    movel([0.641958, -1.476477, -2.502948, -0.732964, 1.570796, 2.212754],accel_mss,speed_ms,0,blend_radius_m)
    movel([0.641515, -1.476223, -2.503164, -0.733002, 1.570796, 2.212311],accel_mss,speed_ms,0,blend_radius_m)
    movel([0.640075, -1.474344, -2.504756, -0.733289, 1.570796, 2.210872],accel_mss,speed_ms,0,blend_radius_m)
    movel([0.638982, -1.472230, -2.506541, -0.733619, 1.570796, 2.209778],accel_mss,speed_ms,0,blend_radius_m)
    movel([0.638629, -1.472579, -2.506246, -0.733564, 1.570796, 2.209425],accel_mss,speed_ms,0,blend_radius_m)
    movel([0.638365, -1.472967, -2.505919, -0.733503, 1.570796, 2.209162],accel_mss,speed_ms,0,blend_radius_m)
    movel([0.638079, -1.473837, -2.505185, -0.733368, 1.570796, 2.208875],accel_mss,speed_ms,0,blend_radius_m)
    movel([0.638058, -1.474782, -2.504385, -0.733222, 1.570796, 2.208855],accel_mss,speed_ms,0,blend_radius_m)
    movel([0.638230, -1.475759, -2.503558, -0.733073, 1.570796, 2.209026],accel_mss,speed_ms,0,blend_radius_m)
    movel([0.638904, -1.477598, -2.501995, -0.732796, 1.570796, 2.209700],accel_mss,speed_ms,0,blend_radius_m)
    movel([0.639570, -1.478960, -2.500835, -0.732594, 1.570796, 2.210367],accel_mss,speed_ms,0,blend_radius_m)
    movel([0.639752, -1.479499, -2.500375, -0.732515, 1.570796, 2.210548],accel_mss,speed_ms,0,blend_radius_m)
    movel([0.639728, -1.479795, -2.500122, -0.732472, 1.570796, 2.210525],accel_mss,speed_ms,0,blend_radius_m)
    movel([0.639572, -1.480098, -2.499864, -0.732428, 1.570796, 2.210369],accel_mss,speed_ms,0,blend_radius_m)
    movel([0.639281, -1.480378, -2.499624, -0.732387, 1.570796, 2.210078],accel_mss,speed_ms,0,blend_radius_m)
    movel([0.638997, -1.480507, -2.499514, -0.732368, 1.570796, 2.209793],accel_mss,speed_ms,0,blend_radius_m)
    movel([0.638451, -1.480478, -2.499539, -0.732373, 1.570796, 2.209248],accel_mss,speed_ms,0,blend_radius_m)
    movel([0.637722, -1.480353, -2.499646, -0.732391, 1.570796, 2.208518],accel_mss,speed_ms,0,blend_radius_m)
    movel([0.637511, -1.480458, -2.499555, -0.732375, 1.570796, 2.208308],accel_mss,speed_ms,0,blend_radius_m)
    movel([0.637299, -1.480720, -2.499332, -0.732338, 1.570796, 2.208095],accel_mss,speed_ms,0,blend_radius_m)
    movel([0.637184, -1.481038, -2.499059, -0.732292, 1.570796, 2.207981],accel_mss,speed_ms,0,blend_radius_m)
    movel([0.637173, -1.481764, -2.498437, -0.732188, 1.570796, 2.207969],accel_mss,speed_ms,0,blend_radius_m)
    movel([0.637454, -1.483028, -2.497352, -0.732009, 1.570796, 2.208251],accel_mss,speed_ms,0,blend_radius_m)
    movel([0.639119, -1.488150, -2.492930, -0.731309, 1.570796, 2.209915],accel_mss,speed_ms,0,blend_radius_m)
    movel([0.639203, -1.488702, -2.492451, -0.731236, 1.570796, 2.209999],accel_mss,speed_ms,0,blend_radius_m)
    movel([0.639148, -1.489297, -2.491934, -0.731158, 1.570796, 2.209944],accel_mss,speed_ms,0,blend_radius_m)
    movel([0.638894, -1.489854, -2.491449, -0.731086, 1.570796, 2.209690],accel_mss,speed_ms,0,blend_radius_m)
    movel([0.638384, -1.490289, -2.491071, -0.731029, 1.570796, 2.209180],accel_mss,speed_ms,0,blend_radius_m)
    movel([0.637804, -1.490445, -2.490935, -0.731009, 1.570796, 2.208600],accel_mss,speed_ms,0,blend_radius_m)
    movel([0.637303, -1.490327, -2.491037, -0.731024, 1.570796, 2.208099],accel_mss,speed_ms,0,blend_radius_m)
    movel([0.636892, -1.490027, -2.491299, -0.731063, 1.570796, 2.207688],accel_mss,speed_ms,0,blend_radius_m)
    movel([0.636580, -1.489644, -2.491632, -0.731113, 1.570796, 2.207376],accel_mss,speed_ms,0,blend_radius_m)
    movel([0.635083, -1.487144, -2.493802, -0.731443, 1.570796, 2.205879],accel_mss,speed_ms,0,blend_radius_m)
    movel([0.633756, -1.484529, -2.496061, -0.731799, 1.570796, 2.204552],accel_mss,speed_ms,0,blend_radius_m)
    movel([0.632600, -1.481802, -2.498404, -0.732182, 1.570796, 2.203396],accel_mss,speed_ms,0,blend_radius_m)
    movel([0.631623, -1.478968, -2.500828, -0.732593, 1.570796, 2.202419],accel_mss,speed_ms,0,blend_radius_m)
    movel([0.631337, -1.477879, -2.501756, -0.732754, 1.570796, 2.202133],accel_mss,speed_ms,0,blend_radius_m)
    movel([0.631258, -1.476708, -2.502752, -0.732929, 1.570796, 2.202055],accel_mss,speed_ms,0,blend_radius_m)
    movel([0.631373, -1.475970, -2.503379, -0.733040, 1.570796, 2.202169],accel_mss,speed_ms,0,blend_radius_m)
    movel([0.631585, -1.475215, -2.504019, -0.733155, 1.570796, 2.202381],accel_mss,speed_ms,0,blend_radius_m)
    movel([0.632182, -1.473679, -2.505318, -0.733392, 1.570796, 2.202978],accel_mss,speed_ms,0,blend_radius_m)
    movel([0.634868, -1.468171, -2.509946, -0.734271, 1.570796, 2.205664],accel_mss,speed_ms,0,blend_radius_m)
    movel([0.635483, -1.466605, -2.511254, -0.734530, 1.570796, 2.206279],accel_mss,speed_ms,0,blend_radius_m)
    movel([0.635855, -1.465194, -2.512429, -0.734766, 1.570796, 2.206652],accel_mss,speed_ms,0,blend_radius_m)
    movel([0.635914, -1.464584, -2.512936, -0.734870, 1.570796, 2.206711],accel_mss,speed_ms,0,blend_radius_m)
    movel([0.635871, -1.464053, -2.513376, -0.734960, 1.570796, 2.206667],accel_mss,speed_ms,0,blend_radius_m)
    movel([0.635709, -1.463622, -2.513734, -0.735033, 1.570796, 2.206506],accel_mss,speed_ms,0,blend_radius_m)
    movel([0.635418, -1.463300, -2.514000, -0.735088, 1.570796, 2.206215],accel_mss,speed_ms,0,blend_radius_m)
    movel([0.634721, -1.462936, -2.514302, -0.735151, 1.570796, 2.205518],accel_mss,speed_ms,0,blend_radius_m)
    movel([0.634424, -1.462720, -2.514481, -0.735188, 1.570796, 2.205220],accel_mss,speed_ms,0,blend_radius_m)
    movel([0.634271, -1.462407, -2.514740, -0.735242, 1.570796, 2.205068],accel_mss,speed_ms,0,blend_radius_m)
    movel([0.634407, -1.461807, -2.515236, -0.735346, 1.570796, 2.205203],accel_mss,speed_ms,0,blend_radius_m)
    movel([0.634800, -1.461179, -2.515754, -0.735456, 1.570796, 2.205597],accel_mss,speed_ms,0,blend_radius_m)
    movel([0.636148, -1.459190, -2.517393, -0.735807, 1.570796, 2.206945],accel_mss,speed_ms,0,blend_radius_m)
    movel([0.637367, -1.457182, -2.519040, -0.736167, 1.570796, 2.208163],accel_mss,speed_ms,0,blend_radius_m)
    movel([0.639488, -1.453116, -2.522357, -0.736916, 1.570796, 2.210284],accel_mss,speed_ms,0,blend_radius_m)
    movel([0.641323, -1.448978, -2.525707, -0.737704, 1.570796, 2.212119],accel_mss,speed_ms,0,blend_radius_m)
    movel([0.643024, -1.444766, -2.529089, -0.738534, 1.570796, 2.213820],accel_mss,speed_ms,0,blend_radius_m)
    speed_ms = 0.005
    movel([0.643024, -1.436436, -2.525376, -0.750577, 1.570796, 2.213820],accel_mss,speed_ms,0,blend_radius_m)
    speed_ms = 0.040
    movel([0.637764, -1.442161, -2.520832, -0.749396, 1.570796, 2.208560],accel_mss,speed_ms,0,blend_radius_m)
    speed_ms = 0.005
    movel([0.637764, -1.450447, -2.524521, -0.737421, 1.570796, 2.208560],accel_mss,speed_ms,0,blend_radius_m)
    speed_ms = 0.025
    movel([0.634464, -1.454408, -2.521306, -0.736675, 1.570796, 2.205260],accel_mss,speed_ms,0,blend_radius_m)
    movel([0.632715, -1.456330, -2.519737, -0.736322, 1.570796, 2.203511],accel_mss,speed_ms,0,blend_radius_m)
    movel([0.630907, -1.458208, -2.518199, -0.735982, 1.570796, 2.201703],accel_mss,speed_ms,0,blend_radius_m)
    movel([0.630497, -1.456900, -2.519271, -0.736218, 1.570796, 2.201294],accel_mss,speed_ms,0,blend_radius_m)
    movel([0.630400, -1.456693, -2.519440, -0.736256, 1.570796, 2.201197],accel_mss,speed_ms,0,blend_radius_m)
    movel([0.630199, -1.456595, -2.519521, -0.736274, 1.570796, 2.200995],accel_mss,speed_ms,0,blend_radius_m)
    movel([0.629906, -1.456693, -2.519440, -0.736256, 1.570796, 2.200702],accel_mss,speed_ms,0,blend_radius_m)
    movel([0.629627, -1.456902, -2.519269, -0.736218, 1.570796, 2.200423],accel_mss,speed_ms,0,blend_radius_m)
    movel([0.627898, -1.458194, -2.518210, -0.735985, 1.570796, 2.198694],accel_mss,speed_ms,0,blend_radius_m)
    movel([0.626047, -1.459278, -2.517320, -0.735791, 1.570796, 2.196843],accel_mss,speed_ms,0,blend_radius_m)
    movel([0.625596, -1.459460, -2.517171, -0.735759, 1.570796, 2.196392],accel_mss,speed_ms,0,blend_radius_m)
    movel([0.625231, -1.459431, -2.517194, -0.735764, 1.570796, 2.196027],accel_mss,speed_ms,0,blend_radius_m)
    movel([0.625146, -1.459173, -2.517406, -0.735810, 1.570796, 2.195943],accel_mss,speed_ms,0,blend_radius_m)
    movel([0.625241, -1.458837, -2.517683, -0.735870, 1.570796, 2.196037],accel_mss,speed_ms,0,blend_radius_m)
    movel([0.626199, -1.456787, -2.519363, -0.736239, 1.570796, 2.196995],accel_mss,speed_ms,0,blend_radius_m)
    movel([0.627476, -1.454770, -2.521011, -0.736608, 1.570796, 2.198272],accel_mss,speed_ms,0,blend_radius_m)
    speed_ms = 0.005
    movel([0.627476, -1.446519, -2.517340, -0.748530, 1.570796, 2.198272],accel_mss,speed_ms,0,blend_radius_m)
    speed_ms = 0.040
    movel([0.627988, -1.451771, -2.513092, -0.747526, 1.570796, 2.198784],accel_mss,speed_ms,0,blend_radius_m)
    speed_ms = 0.005
    movel([0.627988, -1.459981, -2.516742, -0.735666, 1.570796, 2.198784],accel_mss,speed_ms,0,blend_radius_m)
    speed_ms = 0.025
    movel([0.626151, -1.462942, -2.514297, -0.735150, 1.570796, 2.196948],accel_mss,speed_ms,0,blend_radius_m)
    movel([0.625097, -1.464385, -2.513101, -0.734903, 1.570796, 2.195893],accel_mss,speed_ms,0,blend_radius_m)
    movel([0.622748, -1.467165, -2.510787, -0.734437, 1.570796, 2.193545],accel_mss,speed_ms,0,blend_radius_m)
    movel([0.621462, -1.468491, -2.509679, -0.734219, 1.570796, 2.192259],accel_mss,speed_ms,0,blend_radius_m)
    movel([0.618694, -1.470988, -2.507585, -0.733816, 1.570796, 2.189491],accel_mss,speed_ms,0,blend_radius_m)
    movel([0.619378, -1.470024, -2.508394, -0.733970, 1.570796, 2.190174],accel_mss,speed_ms,0,blend_radius_m)
    movel([0.619797, -1.469022, -2.509234, -0.734132, 1.570796, 2.190594],accel_mss,speed_ms,0,blend_radius_m)
    movel([0.619930, -1.468054, -2.510045, -0.734291, 1.570796, 2.190726],accel_mss,speed_ms,0,blend_radius_m)
    movel([0.619753, -1.467190, -2.510766, -0.734433, 1.570796, 2.190549],accel_mss,speed_ms,0,blend_radius_m)
    speed_ms = 0.005
    movel([0.619753, -1.459037, -2.507146, -0.746205, 1.570796, 2.190549],accel_mss,speed_ms,0,blend_radius_m)
    speed_ms = 0.040
    movel([0.608750, -1.458273, -2.507776, -0.746340, 1.570796, 2.179546],accel_mss,speed_ms,0,blend_radius_m)
    speed_ms = 0.005
    movel([0.608750, -1.466431, -2.511399, -0.734559, 1.570796, 2.179546],accel_mss,speed_ms,0,blend_radius_m)
    speed_ms = 0.025
    movel([0.606276, -1.467605, -2.510420, -0.734364, 1.570796, 2.177072],accel_mss,speed_ms,0,blend_radius_m)
    movel([0.603766, -1.468519, -2.509656, -0.734215, 1.570796, 2.174563],accel_mss,speed_ms,0,blend_radius_m)
    movel([0.601263, -1.469162, -2.509117, -0.734110, 1.570796, 2.172059],accel_mss,speed_ms,0,blend_radius_m)
    movel([0.598809, -1.469521, -2.508816, -0.734051, 1.570796, 2.169605],accel_mss,speed_ms,0,blend_radius_m)
    movel([0.599716, -1.468751, -2.509462, -0.734177, 1.570796, 2.170512],accel_mss,speed_ms,0,blend_radius_m)
    movel([0.600486, -1.467955, -2.510127, -0.734307, 1.570796, 2.171283],accel_mss,speed_ms,0,blend_radius_m)
    movel([0.601057, -1.467211, -2.510748, -0.734429, 1.570796, 2.171853],accel_mss,speed_ms,0,blend_radius_m)
    movel([0.601366, -1.466593, -2.511264, -0.734532, 1.570796, 2.172162],accel_mss,speed_ms,0,blend_radius_m)
    movel([0.601345, -1.466181, -2.511607, -0.734601, 1.570796, 2.172142],accel_mss,speed_ms,0,blend_radius_m)
    movel([0.601194, -1.466075, -2.511695, -0.734618, 1.570796, 2.171990],accel_mss,speed_ms,0,blend_radius_m)
    movel([0.600934, -1.466048, -2.511718, -0.734623, 1.570796, 2.171730],accel_mss,speed_ms,0,blend_radius_m)
    movel([0.600067, -1.466274, -2.511529, -0.734585, 1.570796, 2.170864],accel_mss,speed_ms,0,blend_radius_m)
    movel([0.597596, -1.467480, -2.510524, -0.734385, 1.570796, 2.168392],accel_mss,speed_ms,0,blend_radius_m)
    movel([0.596477, -1.467956, -2.510126, -0.734307, 1.570796, 2.167273],accel_mss,speed_ms,0,blend_radius_m)
    movel([0.594203, -1.468674, -2.509526, -0.734189, 1.570796, 2.164999],accel_mss,speed_ms,0,blend_radius_m)
    movel([0.593077, -1.468905, -2.509333, -0.734152, 1.570796, 2.163873],accel_mss,speed_ms,0,blend_radius_m)
    movel([0.591978, -1.469037, -2.509222, -0.734130, 1.570796, 2.162775],accel_mss,speed_ms,0,blend_radius_m)
    movel([0.590919, -1.469071, -2.509194, -0.734125, 1.570796, 2.161716],accel_mss,speed_ms,0,blend_radius_m)
    movel([0.589919, -1.468994, -2.509258, -0.734137, 1.570796, 2.160715],accel_mss,speed_ms,0,blend_radius_m)
    movel([0.591630, -1.468026, -2.510068, -0.734295, 1.570796, 2.162426],accel_mss,speed_ms,0,blend_radius_m)
    movel([0.593324, -1.467014, -2.510913, -0.734462, 1.570796, 2.164121],accel_mss,speed_ms,0,blend_radius_m)
    movel([0.594264, -1.466177, -2.511611, -0.734601, 1.570796, 2.165060],accel_mss,speed_ms,0,blend_radius_m)
    movel([0.595003, -1.465226, -2.512402, -0.734761, 1.570796, 2.165799],accel_mss,speed_ms,0,blend_radius_m)
    movel([0.595149, -1.464828, -2.512733, -0.734828, 1.570796, 2.165945],accel_mss,speed_ms,0,blend_radius_m)
    movel([0.595062, -1.464545, -2.512968, -0.734876, 1.570796, 2.165858],accel_mss,speed_ms,0,blend_radius_m)
    movel([0.594686, -1.464428, -2.513065, -0.734896, 1.570796, 2.165483],accel_mss,speed_ms,0,blend_radius_m)
    movel([0.593960, -1.464526, -2.512983, -0.734879, 1.570796, 2.164756],accel_mss,speed_ms,0,blend_radius_m)
    movel([0.589880, -1.465593, -2.512097, -0.734699, 1.570796, 2.160677],accel_mss,speed_ms,0,blend_radius_m)
    movel([0.587928, -1.465897, -2.511843, -0.734648, 1.570796, 2.158724],accel_mss,speed_ms,0,blend_radius_m)
    movel([0.587015, -1.465903, -2.511839, -0.734647, 1.570796, 2.157811],accel_mss,speed_ms,0,blend_radius_m)
    movel([0.586157, -1.465776, -2.511945, -0.734669, 1.570796, 2.156953],accel_mss,speed_ms,0,blend_radius_m)
    speed_ms = 0.005
    movel([0.586157, -1.457612, -2.508319, -0.746458, 1.570796, 2.156953],accel_mss,speed_ms,0,blend_radius_m)
    speed_ms = 0.040
    movel([0.608445, -1.444545, -2.518925, -0.748919, 1.570796, 2.179242],accel_mss,speed_ms,0,blend_radius_m)
    speed_ms = 0.005
    movel([0.608445, -1.452812, -2.522604, -0.736973, 1.570796, 2.179242],accel_mss,speed_ms,0,blend_radius_m)
    speed_ms = 0.025
    movel([0.609102, -1.451455, -2.523704, -0.737229, 1.570796, 2.179898],accel_mss,speed_ms,0,blend_radius_m)
    movel([0.610004, -1.450153, -2.524759, -0.737478, 1.570796, 2.180800],accel_mss,speed_ms,0,blend_radius_m)
    movel([0.611115, -1.448916, -2.525757, -0.737716, 1.570796, 2.181912],accel_mss,speed_ms,0,blend_radius_m)
    movel([0.612394, -1.447766, -2.526683, -0.737940, 1.570796, 2.183190],accel_mss,speed_ms,0,blend_radius_m)
    movel([0.613809, -1.446716, -2.527526, -0.738146, 1.570796, 2.184605],accel_mss,speed_ms,0,blend_radius_m)
    movel([0.615315, -1.445789, -2.528270, -0.738330, 1.570796, 2.186111],accel_mss,speed_ms,0,blend_radius_m)
    movel([0.616882, -1.444997, -2.528905, -0.738488, 1.570796, 2.187678],accel_mss,speed_ms,0,blend_radius_m)
    movel([0.618464, -1.444359, -2.529414, -0.738615, 1.570796, 2.189261],accel_mss,speed_ms,0,blend_radius_m)
    movel([0.620408, -1.443761, -2.529892, -0.738736, 1.570796, 2.191205],accel_mss,speed_ms,0,blend_radius_m)
    movel([0.624291, -1.442705, -2.530734, -0.738950, 1.570796, 2.195087],accel_mss,speed_ms,0,blend_radius_m)
    movel([0.626231, -1.442020, -2.531280, -0.739089, 1.570796, 2.197028],accel_mss,speed_ms,0,blend_radius_m)
    movel([0.628170, -1.441040, -2.532058, -0.739290, 1.570796, 2.198966],accel_mss,speed_ms,0,blend_radius_m)
    movel([0.629096, -1.440430, -2.532542, -0.739416, 1.570796, 2.199893],accel_mss,speed_ms,0,blend_radius_m)
    movel([0.629958, -1.439753, -2.533079, -0.739557, 1.570796, 2.200754],accel_mss,speed_ms,0,blend_radius_m)
    movel([0.630728, -1.439017, -2.533662, -0.739710, 1.570796, 2.201524],accel_mss,speed_ms,0,blend_radius_m)
    movel([0.631381, -1.438234, -2.534281, -0.739874, 1.570796, 2.202177],accel_mss,speed_ms,0,blend_radius_m)
    movel([0.631884, -1.437414, -2.534928, -0.740047, 1.570796, 2.202680],accel_mss,speed_ms,0,blend_radius_m)
    movel([0.632210, -1.436568, -2.535594, -0.740227, 1.570796, 2.203006],accel_mss,speed_ms,0,blend_radius_m)
    speed_ms = 0.005
    movel([0.632210, -1.428174, -2.531847, -0.752368, 1.570796, 2.203006],accel_mss,speed_ms,0,blend_radius_m)
    speed_ms = 0.040
    movel([0.634472, -1.421241, -2.537198, -0.753950, 1.570796, 2.205268],accel_mss,speed_ms,0,blend_radius_m)
    speed_ms = 0.005
    movel([0.634472, -1.429688, -2.540974, -0.741726, 1.570796, 2.205268],accel_mss,speed_ms,0,blend_radius_m)
    speed_ms = 0.025
    movel([0.630966, -1.434319, -2.537361, -0.740709, 1.570796, 2.201762],accel_mss,speed_ms,0,blend_radius_m)
    movel([0.630012, -1.435247, -2.536633, -0.740509, 1.570796, 2.200808],accel_mss,speed_ms,0,blend_radius_m)
    movel([0.628877, -1.435944, -2.536085, -0.740360, 1.570796, 2.199673],accel_mss,speed_ms,0,blend_radius_m)
    movel([0.627663, -1.436404, -2.535723, -0.740262, 1.570796, 2.198460],accel_mss,speed_ms,0,blend_radius_m)
    movel([0.623784, -1.437426, -2.534919, -0.740045, 1.570796, 2.194581],accel_mss,speed_ms,0,blend_radius_m)
    movel([0.622396, -1.437944, -2.534510, -0.739935, 1.570796, 2.193193],accel_mss,speed_ms,0,blend_radius_m)
    movel([0.621022, -1.438571, -2.534015, -0.739804, 1.570796, 2.191818],accel_mss,speed_ms,0,blend_radius_m)
    movel([0.619676, -1.439294, -2.533443, -0.739652, 1.570796, 2.190472],accel_mss,speed_ms,0,blend_radius_m)
    movel([0.618436, -1.440141, -2.532772, -0.739476, 1.570796, 2.189232],accel_mss,speed_ms,0,blend_radius_m)
    movel([0.617280, -1.441094, -2.532016, -0.739279, 1.570796, 2.188076],accel_mss,speed_ms,0,blend_radius_m)
    movel([0.616136, -1.442049, -2.531256, -0.739083, 1.570796, 2.186932],accel_mss,speed_ms,0,blend_radius_m)
    movel([0.614930, -1.442905, -2.530575, -0.738909, 1.570796, 2.185726],accel_mss,speed_ms,0,blend_radius_m)
    movel([0.615593, -1.439744, -2.533086, -0.739559, 1.570796, 2.186390],accel_mss,speed_ms,0,blend_radius_m)
    movel([0.616059, -1.438916, -2.533742, -0.739731, 1.570796, 2.186855],accel_mss,speed_ms,0,blend_radius_m)
    movel([0.616636, -1.438140, -2.534355, -0.739894, 1.570796, 2.187432],accel_mss,speed_ms,0,blend_radius_m)
    movel([0.617323, -1.437413, -2.534928, -0.740047, 1.570796, 2.188119],accel_mss,speed_ms,0,blend_radius_m)
    movel([0.618129, -1.436734, -2.535464, -0.740191, 1.570796, 2.188926],accel_mss,speed_ms,0,blend_radius_m)
    movel([0.619413, -1.435981, -2.536056, -0.740352, 1.570796, 2.190209],accel_mss,speed_ms,0,blend_radius_m)
    movel([0.621123, -1.435253, -2.536628, -0.740508, 1.570796, 2.191920],accel_mss,speed_ms,0,blend_radius_m)
    movel([0.625153, -1.433842, -2.537735, -0.740812, 1.570796, 2.195949],accel_mss,speed_ms,0,blend_radius_m)
    movel([0.627133, -1.433147, -2.538278, -0.740963, 1.570796, 2.197930],accel_mss,speed_ms,0,blend_radius_m)
    movel([0.628867, -1.432445, -2.538827, -0.741117, 1.570796, 2.199663],accel_mss,speed_ms,0,blend_radius_m)
    movel([0.630181, -1.431732, -2.539383, -0.741273, 1.570796, 2.200977],accel_mss,speed_ms,0,blend_radius_m)
    movel([0.630630, -1.431367, -2.539668, -0.741354, 1.570796, 2.201426],accel_mss,speed_ms,0,blend_radius_m)
    movel([0.630911, -1.430993, -2.539959, -0.741436, 1.570796, 2.201707],accel_mss,speed_ms,0,blend_radius_m)
    speed_ms = 0.005
    movel([0.630911, -1.422556, -2.536188, -0.753645, 1.570796, 2.201707],accel_mss,speed_ms,0,blend_radius_m)
    speed_ms = 0.040
    movel([0.626406, -1.418603, -2.539215, -0.754571, 1.570796, 2.197203],accel_mss,speed_ms,0,blend_radius_m)
    speed_ms = 0.005
    movel([0.626406, -1.427071, -2.543002, -0.742316, 1.570796, 2.197203],accel_mss,speed_ms,0,blend_radius_m)
    speed_ms = 0.025
    movel([0.625978, -1.426676, -2.543308, -0.742406, 1.570796, 2.196775],accel_mss,speed_ms,0,blend_radius_m)
    movel([0.625701, -1.426178, -2.543692, -0.742519, 1.570796, 2.196497],accel_mss,speed_ms,0,blend_radius_m)
    movel([0.625515, -1.424957, -2.544632, -0.742799, 1.570796, 2.196311],accel_mss,speed_ms,0,blend_radius_m)
    movel([0.625692, -1.423549, -2.545715, -0.743125, 1.570796, 2.196488],accel_mss,speed_ms,0,blend_radius_m)
    movel([0.626077, -1.422092, -2.546832, -0.743466, 1.570796, 2.196873],accel_mss,speed_ms,0,blend_radius_m)
    movel([0.626302, -1.421561, -2.547237, -0.743590, 1.570796, 2.197098],accel_mss,speed_ms,0,blend_radius_m)
    movel([0.627024, -1.420869, -2.547766, -0.743754, 1.570796, 2.197820],accel_mss,speed_ms,0,blend_radius_m)
    movel([0.629266, -1.419088, -2.549123, -0.744177, 1.570796, 2.200063],accel_mss,speed_ms,0,blend_radius_m)
    movel([0.633612, -1.415346, -2.551960, -0.745083, 1.570796, 2.204409],accel_mss,speed_ms,0,blend_radius_m)
    movel([0.635707, -1.413393, -2.553432, -0.745564, 1.570796, 2.206503],accel_mss,speed_ms,0,blend_radius_m)
    speed_ms = 0.005
    movel([0.635707, -1.404821, -2.549586, -0.757982, 1.570796, 2.206503],accel_mss,speed_ms,0,blend_radius_m)
    speed_ms = 0.040
    movel([0.631730, -1.404605, -2.549746, -0.758038, 1.570796, 2.202526],accel_mss,speed_ms,0,blend_radius_m)
    speed_ms = 0.005
    movel([0.631730, -1.413178, -2.553593, -0.745617, 1.570796, 2.202526],accel_mss,speed_ms,0,blend_radius_m)
    speed_ms = 0.025
    movel([0.630561, -1.414434, -2.552648, -0.745307, 1.570796, 2.201357],accel_mss,speed_ms,0,blend_radius_m)
    movel([0.629275, -1.415602, -2.551767, -0.745021, 1.570796, 2.200071],accel_mss,speed_ms,0,blend_radius_m)
    movel([0.627884, -1.416569, -2.551035, -0.744785, 1.570796, 2.198680],accel_mss,speed_ms,0,blend_radius_m)
    movel([0.627150, -1.416945, -2.550750, -0.744694, 1.570796, 2.197947],accel_mss,speed_ms,0,blend_radius_m)
    movel([0.625657, -1.417523, -2.550312, -0.744554, 1.570796, 2.196453],accel_mss,speed_ms,0,blend_radius_m)
    movel([0.625143, -1.417996, -2.549953, -0.744440, 1.570796, 2.195940],accel_mss,speed_ms,0,blend_radius_m)
    movel([0.621578, -1.421930, -2.546956, -0.743504, 1.570796, 2.192374],accel_mss,speed_ms,0,blend_radius_m)
    movel([0.621243, -1.422316, -2.546660, -0.743413, 1.570796, 2.192039],accel_mss,speed_ms,0,blend_radius_m)
    movel([0.621016, -1.422721, -2.546349, -0.743318, 1.570796, 2.191812],accel_mss,speed_ms,0,blend_radius_m)
    movel([0.621038, -1.423264, -2.545933, -0.743192, 1.570796, 2.191834],accel_mss,speed_ms,0,blend_radius_m)
    movel([0.621320, -1.423696, -2.545602, -0.743091, 1.570796, 2.192117],accel_mss,speed_ms,0,blend_radius_m)
    movel([0.622190, -1.424884, -2.544689, -0.742816, 1.570796, 2.192987],accel_mss,speed_ms,0,blend_radius_m)
    movel([0.622880, -1.426189, -2.543683, -0.742517, 1.570796, 2.193677],accel_mss,speed_ms,0,blend_radius_m)
    movel([0.623286, -1.427633, -2.542568, -0.742188, 1.570796, 2.194082],accel_mss,speed_ms,0,blend_radius_m)
    movel([0.623292, -1.429238, -2.541324, -0.741827, 1.570796, 2.194088],accel_mss,speed_ms,0,blend_radius_m)
    speed_ms = 0.005
    movel([0.623292, -1.420787, -2.537546, -0.754056, 1.570796, 2.194088],accel_mss,speed_ms,0,blend_radius_m)
    speed_ms = 0.040
    movel([0.614239, -1.430940, -2.529692, -0.751757, 1.570796, 2.185036],accel_mss,speed_ms,0,blend_radius_m)
    speed_ms = 0.005
    movel([0.614239, -1.439312, -2.533428, -0.739649, 1.570796, 2.185036],accel_mss,speed_ms,0,blend_radius_m)
    speed_ms = 0.025
    movel([0.613899, -1.439397, -2.533361, -0.739631, 1.570796, 2.184695],accel_mss,speed_ms,0,blend_radius_m)
    movel([0.613539, -1.439584, -2.533213, -0.739592, 1.570796, 2.184336],accel_mss,speed_ms,0,blend_radius_m)
    movel([0.611897, -1.440794, -2.532254, -0.739341, 1.570796, 2.182693],accel_mss,speed_ms,0,blend_radius_m)
    movel([0.611689, -1.440847, -2.532211, -0.739330, 1.570796, 2.182486],accel_mss,speed_ms,0,blend_radius_m)
    movel([0.611472, -1.440734, -2.532301, -0.739353, 1.570796, 2.182269],accel_mss,speed_ms,0,blend_radius_m)
    movel([0.611391, -1.440464, -2.532516, -0.739409, 1.570796, 2.182188],accel_mss,speed_ms,0,blend_radius_m)
    movel([0.611527, -1.439641, -2.533168, -0.739580, 1.570796, 2.182323],accel_mss,speed_ms,0,blend_radius_m)
    movel([0.612164, -1.438124, -2.534368, -0.739897, 1.570796, 2.182960],accel_mss,speed_ms,0,blend_radius_m)
    movel([0.613130, -1.436783, -2.535425, -0.740181, 1.570796, 2.183926],accel_mss,speed_ms,0,blend_radius_m)
    movel([0.614280, -1.435499, -2.536435, -0.740455, 1.570796, 2.185077],accel_mss,speed_ms,0,blend_radius_m)
    movel([0.615503, -1.434287, -2.537386, -0.740716, 1.570796, 2.186300],accel_mss,speed_ms,0,blend_radius_m)
    movel([0.616788, -1.433202, -2.538236, -0.740951, 1.570796, 2.187584],accel_mss,speed_ms,0,blend_radius_m)
    movel([0.618128, -1.432240, -2.538987, -0.741162, 1.570796, 2.188924],accel_mss,speed_ms,0,blend_radius_m)
    movel([0.619521, -1.431398, -2.539644, -0.741347, 1.570796, 2.190317],accel_mss,speed_ms,0,blend_radius_m)
    movel([0.620965, -1.430671, -2.540210, -0.741508, 1.570796, 2.191761],accel_mss,speed_ms,0,blend_radius_m)
    movel([0.622453, -1.430055, -2.540689, -0.741644, 1.570796, 2.193249],accel_mss,speed_ms,0,blend_radius_m)
    movel([0.623986, -1.429546, -2.541085, -0.741758, 1.570796, 2.194782],accel_mss,speed_ms,0,blend_radius_m)
    movel([0.625558, -1.429138, -2.541401, -0.741849, 1.570796, 2.196355],accel_mss,speed_ms,0,blend_radius_m)
    movel([0.627800, -1.428405, -2.541970, -0.742014, 1.570796, 2.198597],accel_mss,speed_ms,0,blend_radius_m)
    movel([0.630263, -1.427347, -2.542789, -0.742253, 1.570796, 2.201059],accel_mss,speed_ms,0,blend_radius_m)
    movel([0.632999, -1.425997, -2.543831, -0.742561, 1.570796, 2.203795],accel_mss,speed_ms,0,blend_radius_m)
    speed_ms = 0.005
    movel([0.632999, -1.417521, -2.540039, -0.754829, 1.570796, 2.203795],accel_mss,speed_ms,0,blend_radius_m)
    speed_ms = 0.040
    movel([0.631529, -1.416683, -2.540677, -0.755030, 1.570796, 2.202326],accel_mss,speed_ms,0,blend_radius_m)
    speed_ms = 0.005
    movel([0.631529, -1.425165, -2.544473, -0.742752, 1.570796, 2.202326],accel_mss,speed_ms,0,blend_radius_m)
    speed_ms = 0.025
    movel([0.634472, -1.422332, -2.546648, -0.743409, 1.570796, 2.205269],accel_mss,speed_ms,0,blend_radius_m)
    movel([0.637560, -1.419600, -2.548734, -0.744055, 1.570796, 2.208356],accel_mss,speed_ms,0,blend_radius_m)
    movel([0.639176, -1.418327, -2.549702, -0.744360, 1.570796, 2.209972],accel_mss,speed_ms,0,blend_radius_m)
    movel([0.640843, -1.417142, -2.550601, -0.744646, 1.570796, 2.211640],accel_mss,speed_ms,0,blend_radius_m)
    movel([0.642574, -1.416069, -2.551413, -0.744907, 1.570796, 2.213371],accel_mss,speed_ms,0,blend_radius_m)
    movel([0.644367, -1.415131, -2.552122, -0.745136, 1.570796, 2.215163],accel_mss,speed_ms,0,blend_radius_m)
    movel([0.649060, -1.413130, -2.553629, -0.745629, 1.570796, 2.219856],accel_mss,speed_ms,0,blend_radius_m)
    movel([0.651133, -1.412130, -2.554381, -0.745878, 1.570796, 2.221930],accel_mss,speed_ms,0,blend_radius_m)
    movel([0.652150, -1.411557, -2.554810, -0.746021, 1.570796, 2.222947],accel_mss,speed_ms,0,blend_radius_m)
    movel([0.653131, -1.410897, -2.555305, -0.746187, 1.570796, 2.223928],accel_mss,speed_ms,0,blend_radius_m)
    movel([0.655731, -1.408453, -2.557129, -0.746806, 1.570796, 2.226527],accel_mss,speed_ms,0,blend_radius_m)
    speed_ms = 0.005
    movel([0.655731, -1.399844, -2.553262, -0.759283, 1.570796, 2.226527],accel_mss,speed_ms,0,blend_radius_m)
    speed_ms = 0.040
    movel([0.661836, -1.394252, -2.557350, -0.760788, 1.570796, 2.232632],accel_mss,speed_ms,0,blend_radius_m)
    speed_ms = 0.005
    movel([0.661836, -1.402902, -2.561241, -0.748245, 1.570796, 2.232632],accel_mss,speed_ms,0,blend_radius_m)
    speed_ms = 0.025
    movel([0.663890, -1.400838, -2.562759, -0.748792, 1.570796, 2.234687],accel_mss,speed_ms,0,blend_radius_m)
    movel([0.665035, -1.399965, -2.563398, -0.749025, 1.570796, 2.235831],accel_mss,speed_ms,0,blend_radius_m)
    movel([0.666278, -1.399312, -2.563877, -0.749200, 1.570796, 2.237075],accel_mss,speed_ms,0,blend_radius_m)
    movel([0.667177, -1.399037, -2.564078, -0.749274, 1.570796, 2.237974],accel_mss,speed_ms,0,blend_radius_m)
    movel([0.668058, -1.398894, -2.564182, -0.749313, 1.570796, 2.238854],accel_mss,speed_ms,0,blend_radius_m)
    movel([0.669780, -1.398801, -2.564250, -0.749338, 1.570796, 2.240576],accel_mss,speed_ms,0,blend_radius_m)
    movel([0.671376, -1.398578, -2.564413, -0.749398, 1.570796, 2.242173],accel_mss,speed_ms,0,blend_radius_m)
    movel([0.672788, -1.398079, -2.564777, -0.749533, 1.570796, 2.243584],accel_mss,speed_ms,0,blend_radius_m)
    movel([0.675757, -1.396456, -2.565959, -0.749974, 1.570796, 2.246553],accel_mss,speed_ms,0,blend_radius_m)
    movel([0.676370, -1.396174, -2.566165, -0.750051, 1.570796, 2.247166],accel_mss,speed_ms,0,blend_radius_m)
    movel([0.676978, -1.396006, -2.566287, -0.750097, 1.570796, 2.247775],accel_mss,speed_ms,0,blend_radius_m)
    movel([0.678181, -1.395918, -2.566350, -0.750121, 1.570796, 2.248978],accel_mss,speed_ms,0,blend_radius_m)
    movel([0.680510, -1.396020, -2.566276, -0.750093, 1.570796, 2.251307],accel_mss,speed_ms,0,blend_radius_m)
    movel([0.683082, -1.395846, -2.566403, -0.750140, 1.570796, 2.253879],accel_mss,speed_ms,0,blend_radius_m)
    movel([0.684409, -1.395623, -2.566565, -0.750202, 1.570796, 2.255205],accel_mss,speed_ms,0,blend_radius_m)
    movel([0.685767, -1.395218, -2.566859, -0.750313, 1.570796, 2.256564],accel_mss,speed_ms,0,blend_radius_m)
    movel([0.686865, -1.394669, -2.567256, -0.750464, 1.570796, 2.257661],accel_mss,speed_ms,0,blend_radius_m)
    movel([0.687861, -1.393908, -2.567807, -0.750674, 1.570796, 2.258657],accel_mss,speed_ms,0,blend_radius_m)
    movel([0.688550, -1.393039, -2.568435, -0.750915, 1.570796, 2.259346],accel_mss,speed_ms,0,blend_radius_m)
    movel([0.688714, -1.392599, -2.568753, -0.751037, 1.570796, 2.259510],accel_mss,speed_ms,0,blend_radius_m)
    movel([0.688723, -1.392174, -2.569060, -0.751156, 1.570796, 2.259519],accel_mss,speed_ms,0,blend_radius_m)
    movel([0.688416, -1.391422, -2.569601, -0.751366, 1.570796, 2.259212],accel_mss,speed_ms,0,blend_radius_m)
    movel([0.687831, -1.390766, -2.570073, -0.751550, 1.570796, 2.258627],accel_mss,speed_ms,0,blend_radius_m)
    movel([0.687019, -1.390220, -2.570465, -0.751704, 1.570796, 2.257815],accel_mss,speed_ms,0,blend_radius_m)
    movel([0.686046, -1.389794, -2.570771, -0.751824, 1.570796, 2.256842],accel_mss,speed_ms,0,blend_radius_m)
    movel([0.684965, -1.389510, -2.570975, -0.751904, 1.570796, 2.255761],accel_mss,speed_ms,0,blend_radius_m)
    movel([0.683839, -1.389375, -2.571072, -0.751943, 1.570796, 2.254635],accel_mss,speed_ms,0,blend_radius_m)
    movel([0.682724, -1.389408, -2.571048, -0.751933, 1.570796, 2.253520],accel_mss,speed_ms,0,blend_radius_m)
    movel([0.681679, -1.389620, -2.570896, -0.751873, 1.570796, 2.252475],accel_mss,speed_ms,0,blend_radius_m)
    movel([0.680107, -1.390284, -2.570419, -0.751686, 1.570796, 2.250903],accel_mss,speed_ms,0,blend_radius_m)
    movel([0.675473, -1.392714, -2.568670, -0.751005, 1.570796, 2.246269],accel_mss,speed_ms,0,blend_radius_m)
    movel([0.672351, -1.394092, -2.567674, -0.750623, 1.570796, 2.243147],accel_mss,speed_ms,0,blend_radius_m)
    movel([0.669641, -1.394935, -2.567064, -0.750390, 1.570796, 2.240437],accel_mss,speed_ms,0,blend_radius_m)
    movel([0.668305, -1.395322, -2.566783, -0.750284, 1.570796, 2.239101],accel_mss,speed_ms,0,blend_radius_m)
    movel([0.666980, -1.395830, -2.566414, -0.750145, 1.570796, 2.237776],accel_mss,speed_ms,0,blend_radius_m)
    movel([0.665633, -1.396532, -2.565904, -0.749953, 1.570796, 2.236430],accel_mss,speed_ms,0,blend_radius_m)
    movel([0.664346, -1.397350, -2.565309, -0.749730, 1.570796, 2.235142],accel_mss,speed_ms,0,blend_radius_m)
    movel([0.663112, -1.398265, -2.564641, -0.749482, 1.570796, 2.233909],accel_mss,speed_ms,0,blend_radius_m)
    movel([0.661932, -1.399254, -2.563919, -0.749216, 1.570796, 2.232728],accel_mss,speed_ms,0,blend_radius_m)
    movel([0.659712, -1.401374, -2.562365, -0.748649, 1.570796, 2.230508],accel_mss,speed_ms,0,blend_radius_m)
    movel([0.657647, -1.403546, -2.560767, -0.748076, 1.570796, 2.228444],accel_mss,speed_ms,0,blend_radius_m)
    speed_ms = 0.005
    movel([0.657647, -1.394900, -2.556878, -0.760611, 1.570796, 2.228444],accel_mss,speed_ms,0,blend_radius_m)
    speed_ms = 0.040
    movel([0.654415, -1.395213, -2.556651, -0.760526, 1.570796, 2.225212],accel_mss,speed_ms,0,blend_radius_m)
    speed_ms = 0.005
    movel([0.654415, -1.403856, -2.560538, -0.747995, 1.570796, 2.225212],accel_mss,speed_ms,0,blend_radius_m)
    speed_ms = 0.025
    movel([0.657764, -1.400491, -2.563013, -0.748885, 1.570796, 2.228560],accel_mss,speed_ms,0,blend_radius_m)
    movel([0.659213, -1.399123, -2.564014, -0.749251, 1.570796, 2.230010],accel_mss,speed_ms,0,blend_radius_m)
    movel([0.660598, -1.397708, -2.565048, -0.749633, 1.570796, 2.231394],accel_mss,speed_ms,0,blend_radius_m)
    movel([0.661658, -1.396409, -2.565994, -0.749987, 1.570796, 2.232454],accel_mss,speed_ms,0,blend_radius_m)
    movel([0.662556, -1.395052, -2.566979, -0.750358, 1.570796, 2.233353],accel_mss,speed_ms,0,blend_radius_m)
    movel([0.663277, -1.393664, -2.567984, -0.750741, 1.570796, 2.234073],accel_mss,speed_ms,0,blend_radius_m)
    movel([0.663803, -1.392274, -2.568987, -0.751128, 1.570796, 2.234600],accel_mss,speed_ms,0,blend_radius_m)
    movel([0.664421, -1.392300, -2.568969, -0.751120, 1.570796, 2.235217],accel_mss,speed_ms,0,blend_radius_m)
    movel([0.664952, -1.392477, -2.568841, -0.751071, 1.570796, 2.235749],accel_mss,speed_ms,0,blend_radius_m)
    movel([0.665902, -1.393010, -2.568456, -0.750923, 1.570796, 2.236698],accel_mss,speed_ms,0,blend_radius_m)
    movel([0.666957, -1.393447, -2.568141, -0.750801, 1.570796, 2.237753],accel_mss,speed_ms,0,blend_radius_m)
    movel([0.667567, -1.393492, -2.568108, -0.750789, 1.570796, 2.238364],accel_mss,speed_ms,0,blend_radius_m)
    movel([0.668235, -1.393324, -2.568229, -0.750835, 1.570796, 2.239032],accel_mss,speed_ms,0,blend_radius_m)
    movel([0.676287, -1.390042, -2.570593, -0.751754, 1.570796, 2.247083],accel_mss,speed_ms,0,blend_radius_m)
    movel([0.676745, -1.389077, -2.571285, -0.752027, 1.570796, 2.247541],accel_mss,speed_ms,0,blend_radius_m)
    movel([0.676931, -1.388102, -2.571983, -0.752304, 1.570796, 2.247728],accel_mss,speed_ms,0,blend_radius_m)
    movel([0.676838, -1.387168, -2.572650, -0.752571, 1.570796, 2.247634],accel_mss,speed_ms,0,blend_radius_m)
    movel([0.676462, -1.386329, -2.573248, -0.752812, 1.570796, 2.247259],accel_mss,speed_ms,0,blend_radius_m)
    movel([0.677727, -1.386688, -2.572992, -0.752709, 1.570796, 2.248523],accel_mss,speed_ms,0,blend_radius_m)
    movel([0.678785, -1.387289, -2.572563, -0.752536, 1.570796, 2.249582],accel_mss,speed_ms,0,blend_radius_m)
    movel([0.679587, -1.388095, -2.571987, -0.752306, 1.570796, 2.250383],accel_mss,speed_ms,0,blend_radius_m)
    movel([0.680086, -1.389070, -2.571290, -0.752029, 1.570796, 2.250882],accel_mss,speed_ms,0,blend_radius_m)
    speed_ms = 0.005
    movel([0.680086, -1.380317, -2.567338, -0.764734, 1.570796, 2.250882],accel_mss,speed_ms,0,blend_radius_m)
    speed_ms = 0.040
    movel([0.682625, -1.376904, -2.569742, -0.765743, 1.570796, 2.253421],accel_mss,speed_ms,0,blend_radius_m)
    speed_ms = 0.005
    movel([0.682625, -1.385682, -2.573709, -0.752998, 1.570796, 2.253421],accel_mss,speed_ms,0,blend_radius_m)
    speed_ms = 0.025
    movel([0.684185, -1.384026, -2.574885, -0.753478, 1.570796, 2.254981],accel_mss,speed_ms,0,blend_radius_m)
    movel([0.685568, -1.382373, -2.576055, -0.753961, 1.570796, 2.256364],accel_mss,speed_ms,0,blend_radius_m)
    movel([0.686790, -1.380715, -2.577224, -0.754450, 1.570796, 2.257586],accel_mss,speed_ms,0,blend_radius_m)
    movel([0.687866, -1.379044, -2.578399, -0.754946, 1.570796, 2.258662],accel_mss,speed_ms,0,blend_radius_m)
    movel([0.688814, -1.377349, -2.579586, -0.755454, 1.570796, 2.259610],accel_mss,speed_ms,0,blend_radius_m)
    movel([0.689650, -1.375618, -2.580795, -0.755976, 1.570796, 2.260446],accel_mss,speed_ms,0,blend_radius_m)
    movel([0.691053, -1.372013, -2.583298, -0.757078, 1.570796, 2.261849],accel_mss,speed_ms,0,blend_radius_m)
    movel([0.685784, -1.377783, -2.579283, -0.755323, 1.570796, 2.256581],accel_mss,speed_ms,0,blend_radius_m)
    movel([0.686315, -1.377115, -2.579750, -0.755524, 1.570796, 2.257112],accel_mss,speed_ms,0,blend_radius_m)
    movel([0.686734, -1.376414, -2.580240, -0.755735, 1.570796, 2.257530],accel_mss,speed_ms,0,blend_radius_m)
    movel([0.687266, -1.374941, -2.581266, -0.756182, 1.570796, 2.258063],accel_mss,speed_ms,0,blend_radius_m)
    movel([0.687446, -1.373417, -2.582325, -0.756647, 1.570796, 2.258243],accel_mss,speed_ms,0,blend_radius_m)
    movel([0.687344, -1.371902, -2.583375, -0.757112, 1.570796, 2.258140],accel_mss,speed_ms,0,blend_radius_m)
    movel([0.687026, -1.370449, -2.584378, -0.757562, 1.570796, 2.257822],accel_mss,speed_ms,0,blend_radius_m)
    movel([0.686563, -1.369120, -2.585293, -0.757976, 1.570796, 2.257359],accel_mss,speed_ms,0,blend_radius_m)
    movel([0.685474, -1.367060, -2.586706, -0.758623, 1.570796, 2.256271],accel_mss,speed_ms,0,blend_radius_m)
    movel([0.684812, -1.370325, -2.584463, -0.757601, 1.570796, 2.255609],accel_mss,speed_ms,0,blend_radius_m)
    movel([0.684211, -1.372020, -2.583293, -0.757076, 1.570796, 2.255007],accel_mss,speed_ms,0,blend_radius_m)
    movel([0.683325, -1.373573, -2.582217, -0.756599, 1.570796, 2.254122],accel_mss,speed_ms,0,blend_radius_m)
    movel([0.682679, -1.373073, -2.582564, -0.756752, 1.570796, 2.253475],accel_mss,speed_ms,0,blend_radius_m)
    movel([0.682168, -1.372424, -2.583013, -0.756952, 1.570796, 2.252964],accel_mss,speed_ms,0,blend_radius_m)
    movel([0.681364, -1.370863, -2.584092, -0.757434, 1.570796, 2.252160],accel_mss,speed_ms,0,blend_radius_m)
    movel([0.680547, -1.369256, -2.585199, -0.757934, 1.570796, 2.251343],accel_mss,speed_ms,0,blend_radius_m)
    movel([0.680018, -1.368550, -2.585684, -0.758154, 1.570796, 2.250814],accel_mss,speed_ms,0,blend_radius_m)
    movel([0.679351, -1.367971, -2.586082, -0.758336, 1.570796, 2.250148],accel_mss,speed_ms,0,blend_radius_m)
    movel([0.677808, -1.369363, -2.585126, -0.757900, 1.570796, 2.248604],accel_mss,speed_ms,0,blend_radius_m)
    movel([0.676519, -1.370920, -2.584053, -0.757416, 1.570796, 2.247316],accel_mss,speed_ms,0,blend_radius_m)
    movel([0.675488, -1.370319, -2.584467, -0.757603, 1.570796, 2.246284],accel_mss,speed_ms,0,blend_radius_m)
    movel([0.674651, -1.369527, -2.585013, -0.757849, 1.570796, 2.245448],accel_mss,speed_ms,0,blend_radius_m)
    movel([0.674028, -1.368559, -2.585679, -0.758152, 1.570796, 2.244825],accel_mss,speed_ms,0,blend_radius_m)
    movel([0.673638, -1.367440, -2.586446, -0.758503, 1.570796, 2.244435],accel_mss,speed_ms,0,blend_radius_m)
    movel([0.673439, -1.367540, -2.586377, -0.758472, 1.570796, 2.244235],accel_mss,speed_ms,0,blend_radius_m)
    movel([0.671420, -1.369210, -2.585231, -0.757948, 1.570796, 2.242217],accel_mss,speed_ms,0,blend_radius_m)
    movel([0.668987, -1.371379, -2.583736, -0.757274, 1.570796, 2.239783],accel_mss,speed_ms,0,blend_radius_m)
    movel([0.667931, -1.372523, -2.582945, -0.756921, 1.570796, 2.238728],accel_mss,speed_ms,0,blend_radius_m)
    movel([0.667041, -1.373636, -2.582173, -0.756580, 1.570796, 2.237837],accel_mss,speed_ms,0,blend_radius_m)
    movel([0.665423, -1.376052, -2.580492, -0.755845, 1.570796, 2.236220],accel_mss,speed_ms,0,blend_radius_m)
    movel([0.664409, -1.371628, -2.583564, -0.757197, 1.570796, 2.235205],accel_mss,speed_ms,0,blend_radius_m)
    movel([0.663251, -1.372803, -2.582751, -0.756835, 1.570796, 2.234047],accel_mss,speed_ms,0,blend_radius_m)
    movel([0.662173, -1.374044, -2.581890, -0.756455, 1.570796, 2.232970],accel_mss,speed_ms,0,blend_radius_m)
    movel([0.660249, -1.376663, -2.580066, -0.755660, 1.570796, 2.231045],accel_mss,speed_ms,0,blend_radius_m)
    movel([0.658646, -1.379356, -2.578180, -0.754853, 1.570796, 2.229442],accel_mss,speed_ms,0,blend_radius_m)
    movel([0.656967, -1.382805, -2.575749, -0.753835, 1.570796, 2.227763],accel_mss,speed_ms,0,blend_radius_m)
    movel([0.656689, -1.383176, -2.575487, -0.753726, 1.570796, 2.227485],accel_mss,speed_ms,0,blend_radius_m)
    movel([0.656331, -1.383488, -2.575266, -0.753635, 1.570796, 2.227127],accel_mss,speed_ms,0,blend_radius_m)
    movel([0.655764, -1.383746, -2.575083, -0.753560, 1.570796, 2.226561],accel_mss,speed_ms,0,blend_radius_m)
    movel([0.652053, -1.384374, -2.574638, -0.753377, 1.570796, 2.222849],accel_mss,speed_ms,0,blend_radius_m)
    movel([0.650268, -1.384420, -2.574605, -0.753364, 1.570796, 2.221064],accel_mss,speed_ms,0,blend_radius_m)
    movel([0.649684, -1.384265, -2.574715, -0.753409, 1.570796, 2.220481],accel_mss,speed_ms,0,blend_radius_m)
    movel([0.649446, -1.383943, -2.574943, -0.753502, 1.570796, 2.220242],accel_mss,speed_ms,0,blend_radius_m)
    movel([0.649853, -1.386388, -2.573206, -0.752795, 1.570796, 2.220650],accel_mss,speed_ms,0,blend_radius_m)
    movel([0.650227, -1.387521, -2.572398, -0.752470, 1.570796, 2.221024],accel_mss,speed_ms,0,blend_radius_m)
    movel([0.650709, -1.388588, -2.571635, -0.752166, 1.570796, 2.221505],accel_mss,speed_ms,0,blend_radius_m)
    movel([0.647029, -1.390275, -2.570426, -0.751688, 1.570796, 2.217825],accel_mss,speed_ms,0,blend_radius_m)
    movel([0.643033, -1.392287, -2.568978, -0.751124, 1.570796, 2.213829],accel_mss,speed_ms,0,blend_radius_m)
    movel([0.641066, -1.393410, -2.568167, -0.750812, 1.570796, 2.211862],accel_mss,speed_ms,0,blend_radius_m)
    movel([0.639201, -1.394601, -2.567305, -0.750482, 1.570796, 2.209997],accel_mss,speed_ms,0,blend_radius_m)
    movel([0.637498, -1.395863, -2.566390, -0.750136, 1.570796, 2.208294],accel_mss,speed_ms,0,blend_radius_m)
    movel([0.636017, -1.397186, -2.565428, -0.749775, 1.570796, 2.206814],accel_mss,speed_ms,0,blend_radius_m)
    movel([0.637602, -1.396805, -2.565705, -0.749878, 1.570796, 2.208398],accel_mss,speed_ms,0,blend_radius_m)
    movel([0.639142, -1.396591, -2.565861, -0.749937, 1.570796, 2.209939],accel_mss,speed_ms,0,blend_radius_m)
    movel([0.640615, -1.396559, -2.565884, -0.749946, 1.570796, 2.211411],accel_mss,speed_ms,0,blend_radius_m)
    movel([0.642003, -1.396730, -2.565760, -0.749899, 1.570796, 2.212799],accel_mss,speed_ms,0,blend_radius_m)
    movel([0.640831, -1.397176, -2.565436, -0.749778, 1.570796, 2.211628],accel_mss,speed_ms,0,blend_radius_m)
    movel([0.638537, -1.398337, -2.564589, -0.749463, 1.570796, 2.209333],accel_mss,speed_ms,0,blend_radius_m)
    movel([0.637430, -1.399041, -2.564075, -0.749273, 1.570796, 2.208227],accel_mss,speed_ms,0,blend_radius_m)
    movel([0.635360, -1.400650, -2.562897, -0.748842, 1.570796, 2.206157],accel_mss,speed_ms,0,blend_radius_m)
    movel([0.634413, -1.401543, -2.562241, -0.748605, 1.570796, 2.205210],accel_mss,speed_ms,0,blend_radius_m)
    movel([0.633542, -1.402484, -2.561549, -0.748356, 1.570796, 2.204338],accel_mss,speed_ms,0,blend_radius_m)
    speed_ms = 0.005
    movel([0.633542, -1.393830, -2.557656, -0.760903, 1.570796, 2.204338],accel_mss,speed_ms,0,blend_radius_m)
    speed_ms = 0.040
    movel([0.636386, -1.399066, -2.553833, -0.759490, 1.570796, 2.207182],accel_mss,speed_ms,0,blend_radius_m)
    speed_ms = 0.005
    movel([0.636386, -1.407681, -2.557704, -0.747004, 1.570796, 2.207182],accel_mss,speed_ms,0,blend_radius_m)
    speed_ms = 0.025
    movel([0.637314, -1.406280, -2.558745, -0.747364, 1.570796, 2.208111],accel_mss,speed_ms,0,blend_radius_m)
    movel([0.638362, -1.404895, -2.559771, -0.747724, 1.570796, 2.209158],accel_mss,speed_ms,0,blend_radius_m)
    movel([0.639519, -1.403542, -2.560770, -0.748077, 1.570796, 2.210315],accel_mss,speed_ms,0,blend_radius_m)
    movel([0.640773, -1.402239, -2.561729, -0.748420, 1.570796, 2.211570],accel_mss,speed_ms,0,blend_radius_m)
    movel([0.642119, -1.401000, -2.562640, -0.748749, 1.570796, 2.212915],accel_mss,speed_ms,0,blend_radius_m)
    movel([0.643542, -1.399840, -2.563490, -0.749059, 1.570796, 2.214339],accel_mss,speed_ms,0,blend_radius_m)
    movel([0.645035, -1.398773, -2.564271, -0.749345, 1.570796, 2.215832],accel_mss,speed_ms,0,blend_radius_m)
    movel([0.646587, -1.397817, -2.564968, -0.749604, 1.570796, 2.217384],accel_mss,speed_ms,0,blend_radius_m)
    movel([0.651504, -1.395060, -2.566973, -0.750356, 1.570796, 2.222301],accel_mss,speed_ms,0,blend_radius_m)
    movel([0.652584, -1.394320, -2.567509, -0.750560, 1.570796, 2.223380],accel_mss,speed_ms,0,blend_radius_m)
    movel([0.653628, -1.393474, -2.568121, -0.750794, 1.570796, 2.224424],accel_mss,speed_ms,0,blend_radius_m)
    movel([0.654647, -1.392483, -2.568837, -0.751069, 1.570796, 2.225443],accel_mss,speed_ms,0,blend_radius_m)
    movel([0.655657, -1.391300, -2.569689, -0.751400, 1.570796, 2.226453],accel_mss,speed_ms,0,blend_radius_m)
    movel([0.658245, -1.387723, -2.572253, -0.752412, 1.570796, 2.229042],accel_mss,speed_ms,0,blend_radius_m)
    movel([0.659612, -1.385970, -2.573503, -0.752915, 1.570796, 2.230408],accel_mss,speed_ms,0,blend_radius_m)
    movel([0.661189, -1.384329, -2.574670, -0.753390, 1.570796, 2.231986],accel_mss,speed_ms,0,blend_radius_m)
    movel([0.662268, -1.383437, -2.575302, -0.753650, 1.570796, 2.233065],accel_mss,speed_ms,0,blend_radius_m)
    movel([0.663410, -1.382641, -2.575865, -0.753883, 1.570796, 2.234206],accel_mss,speed_ms,0,blend_radius_m)
    movel([0.665831, -1.381298, -2.576813, -0.754277, 1.570796, 2.236627],accel_mss,speed_ms,0,blend_radius_m)
    movel([0.668358, -1.380204, -2.577584, -0.754601, 1.570796, 2.239154],accel_mss,speed_ms,0,blend_radius_m)
    movel([0.670899, -1.379264, -2.578245, -0.754881, 1.570796, 2.241695],accel_mss,speed_ms,0,blend_radius_m)
    movel([0.673349, -1.378439, -2.578823, -0.755127, 1.570796, 2.244146],accel_mss,speed_ms,0,blend_radius_m)
    movel([0.675779, -1.377820, -2.579257, -0.755312, 1.570796, 2.246575],accel_mss,speed_ms,0,blend_radius_m)
    movel([0.676936, -1.377654, -2.579373, -0.755362, 1.570796, 2.247732],accel_mss,speed_ms,0,blend_radius_m)
    movel([0.678032, -1.377616, -2.579400, -0.755373, 1.570796, 2.248829],accel_mss,speed_ms,0,blend_radius_m)
    movel([0.679041, -1.377734, -2.579317, -0.755338, 1.570796, 2.249838],accel_mss,speed_ms,0,blend_radius_m)
    movel([0.679953, -1.378031, -2.579109, -0.755249, 1.570796, 2.250749],accel_mss,speed_ms,0,blend_radius_m)
    speed_ms = 0.005
    movel([0.679953, -1.369198, -2.575109, -0.768082, 1.570796, 2.250749],accel_mss,speed_ms,0,blend_radius_m)
    speed_ms = 0.040
    movel([0.680324, -1.370938, -2.573904, -0.767547, 1.570796, 2.251120],accel_mss,speed_ms,0,blend_radius_m)
    speed_ms = 0.005
    movel([0.680324, -1.379759, -2.577897, -0.754733, 1.570796, 2.251120],accel_mss,speed_ms,0,blend_radius_m)
    speed_ms = 0.025
    movel([0.680472, -1.380248, -2.577553, -0.754588, 1.570796, 2.251269],accel_mss,speed_ms,0,blend_radius_m)
    movel([0.680607, -1.381026, -2.577005, -0.754358, 1.570796, 2.251403],accel_mss,speed_ms,0,blend_radius_m)
    movel([0.680415, -1.382962, -2.575638, -0.753789, 1.570796, 2.251212],accel_mss,speed_ms,0,blend_radius_m)
    movel([0.680140, -1.383978, -2.574919, -0.753492, 1.570796, 2.250936],accel_mss,speed_ms,0,blend_radius_m)
    movel([0.679886, -1.384452, -2.574583, -0.753355, 1.570796, 2.250682],accel_mss,speed_ms,0,blend_radius_m)
    movel([0.679748, -1.384511, -2.574541, -0.753337, 1.570796, 2.250544],accel_mss,speed_ms,0,blend_radius_m)
    movel([0.679605, -1.384387, -2.574628, -0.753373, 1.570796, 2.250401],accel_mss,speed_ms,0,blend_radius_m)
    movel([0.678556, -1.382444, -2.576005, -0.753941, 1.570796, 2.249352],accel_mss,speed_ms,0,blend_radius_m)
    movel([0.677827, -1.381621, -2.576586, -0.754182, 1.570796, 2.248623],accel_mss,speed_ms,0,blend_radius_m)
    movel([0.677344, -1.381336, -2.576787, -0.754266, 1.570796, 2.248140],accel_mss,speed_ms,0,blend_radius_m)
    movel([0.676759, -1.381163, -2.576909, -0.754317, 1.570796, 2.247556],accel_mss,speed_ms,0,blend_radius_m)
    movel([0.676002, -1.381140, -2.576925, -0.754324, 1.570796, 2.246799],accel_mss,speed_ms,0,blend_radius_m)
    movel([0.675193, -1.381241, -2.576854, -0.754294, 1.570796, 2.245989],accel_mss,speed_ms,0,blend_radius_m)
    movel([0.673139, -1.381692, -2.576535, -0.754161, 1.570796, 2.243936],accel_mss,speed_ms,0,blend_radius_m)
    movel([0.671022, -1.382358, -2.576065, -0.753966, 1.570796, 2.241819],accel_mss,speed_ms,0,blend_radius_m)
    movel([0.668907, -1.383214, -2.575460, -0.753715, 1.570796, 2.239703],accel_mss,speed_ms,0,blend_radius_m)
    movel([0.666865, -1.384233, -2.574738, -0.753418, 1.570796, 2.237662],accel_mss,speed_ms,0,blend_radius_m)
    movel([0.666548, -1.386886, -2.572851, -0.752652, 1.570796, 2.237345],accel_mss,speed_ms,0,blend_radius_m)
    movel([0.665908, -1.389602, -2.570908, -0.751878, 1.570796, 2.236704],accel_mss,speed_ms,0,blend_radius_m)
    movel([0.665535, -1.388831, -2.571461, -0.752097, 1.570796, 2.236331],accel_mss,speed_ms,0,blend_radius_m)
    movel([0.664970, -1.388198, -2.571914, -0.752277, 1.570796, 2.235766],accel_mss,speed_ms,0,blend_radius_m)
    movel([0.664228, -1.387728, -2.572250, -0.752411, 1.570796, 2.235024],accel_mss,speed_ms,0,blend_radius_m)
    movel([0.663335, -1.387437, -2.572458, -0.752494, 1.570796, 2.234131],accel_mss,speed_ms,0,blend_radius_m)
    movel([0.662824, -1.387478, -2.572429, -0.752482, 1.570796, 2.233620],accel_mss,speed_ms,0,blend_radius_m)
    movel([0.662439, -1.387841, -2.572169, -0.752379, 1.570796, 2.233236],accel_mss,speed_ms,0,blend_radius_m)
    movel([0.659039, -1.392277, -2.568985, -0.751127, 1.570796, 2.229836],accel_mss,speed_ms,0,blend_radius_m)
    movel([0.657166, -1.394455, -2.567412, -0.750523, 1.570796, 2.227962],accel_mss,speed_ms,0,blend_radius_m)
    movel([0.655132, -1.396589, -2.565863, -0.749938, 1.570796, 2.225928],accel_mss,speed_ms,0,blend_radius_m)
    movel([0.652972, -1.398610, -2.564390, -0.749389, 1.570796, 2.223768],accel_mss,speed_ms,0,blend_radius_m)
    movel([0.650715, -1.400452, -2.563042, -0.748895, 1.570796, 2.221511],accel_mss,speed_ms,0,blend_radius_m)
    movel([0.646073, -1.404040, -2.560402, -0.747947, 1.570796, 2.216869],accel_mss,speed_ms,0,blend_radius_m)
    movel([0.643941, -1.405968, -2.558976, -0.747445, 1.570796, 2.214738],accel_mss,speed_ms,0,blend_radius_m)
    movel([0.642036, -1.408099, -2.557393, -0.746897, 1.570796, 2.212832],accel_mss,speed_ms,0,blend_radius_m)
    speed_ms = 0.005
    movel([0.642036, -1.399487, -2.553524, -0.759378, 1.570796, 2.212832],accel_mss,speed_ms,0,blend_radius_m)
    speed_ms = 0.040
    movel([0.652406, -1.400382, -2.552866, -0.759141, 1.570796, 2.223202],accel_mss,speed_ms,0,blend_radius_m)
    speed_ms = 0.005
    movel([0.652406, -1.408988, -2.556731, -0.746670, 1.570796, 2.223202],accel_mss,speed_ms,0,blend_radius_m)
    speed_ms = 0.025
    movel([0.650892, -1.410707, -2.555447, -0.746235, 1.570796, 2.221688],accel_mss,speed_ms,0,blend_radius_m)
    movel([0.649148, -1.412267, -2.554278, -0.745844, 1.570796, 2.219944],accel_mss,speed_ms,0,blend_radius_m)
    movel([0.647232, -1.413618, -2.553262, -0.745508, 1.570796, 2.218028],accel_mss,speed_ms,0,blend_radius_m)
    movel([0.645203, -1.414719, -2.552433, -0.745237, 1.570796, 2.216000],accel_mss,speed_ms,0,blend_radius_m)
    speed_ms = 0.005
    movel([0.645203, -1.406157, -2.548592, -0.757639, 1.570796, 2.216000],accel_mss,speed_ms,0,blend_radius_m)
    speed_ms = 0.040
    movel([0.644708, -1.402598, -2.551232, -0.758559, 1.570796, 2.215504],accel_mss,speed_ms,0,blend_radius_m)
    speed_ms = 0.005
    movel([0.644708, -1.411187, -2.555088, -0.746114, 1.570796, 2.215504],accel_mss,speed_ms,0,blend_radius_m)
    speed_ms = 0.025
    movel([0.632928, -1.420166, -2.548302, -0.743920, 1.570796, 2.203724],accel_mss,speed_ms,0,blend_radius_m)
    movel([0.632254, -1.420811, -2.547810, -0.743767, 1.570796, 2.203050],accel_mss,speed_ms,0,blend_radius_m)
    movel([0.631894, -1.421742, -2.547099, -0.743548, 1.570796, 2.202690],accel_mss,speed_ms,0,blend_radius_m)
    movel([0.631428, -1.422941, -2.546181, -0.743267, 1.570796, 2.202224],accel_mss,speed_ms,0,blend_radius_m)
    movel([0.630697, -1.424121, -2.545275, -0.742992, 1.570796, 2.201494],accel_mss,speed_ms,0,blend_radius_m)
    speed_ms = 0.005
    movel([0.630697, -1.415631, -2.541475, -0.755283, 1.570796, 2.201494],accel_mss,speed_ms,0,blend_radius_m)
    speed_ms = 0.040
    movel([0.643692, -1.414403, -2.542405, -0.755581, 1.570796, 2.214488],accel_mss,speed_ms,0,blend_radius_m)
    speed_ms = 0.005
    movel([0.643692, -1.422902, -2.546211, -0.743276, 1.570796, 2.214488],accel_mss,speed_ms,0,blend_radius_m)
    speed_ms = 0.025
    movel([0.644486, -1.421667, -2.547157, -0.743566, 1.570796, 2.215283],accel_mss,speed_ms,0,blend_radius_m)
    movel([0.645426, -1.420470, -2.548071, -0.743848, 1.570796, 2.216222],accel_mss,speed_ms,0,blend_radius_m)
    movel([0.646493, -1.419333, -2.548937, -0.744119, 1.570796, 2.217289],accel_mss,speed_ms,0,blend_radius_m)
    movel([0.647675, -1.418273, -2.549743, -0.744373, 1.570796, 2.218471],accel_mss,speed_ms,0,blend_radius_m)
    movel([0.648555, -1.417600, -2.550254, -0.744535, 1.570796, 2.219351],accel_mss,speed_ms,0,blend_radius_m)
    movel([0.649486, -1.417003, -2.550706, -0.744680, 1.570796, 2.220283],accel_mss,speed_ms,0,blend_radius_m)
    movel([0.650446, -1.416529, -2.551066, -0.744795, 1.570796, 2.221242],accel_mss,speed_ms,0,blend_radius_m)
    movel([0.651421, -1.416216, -2.551302, -0.744871, 1.570796, 2.222217],accel_mss,speed_ms,0,blend_radius_m)
    movel([0.652201, -1.416139, -2.551360, -0.744889, 1.570796, 2.222997],accel_mss,speed_ms,0,blend_radius_m)
    movel([0.652960, -1.416240, -2.551284, -0.744865, 1.570796, 2.223756],accel_mss,speed_ms,0,blend_radius_m)
    movel([0.653689, -1.416481, -2.551102, -0.744806, 1.570796, 2.224486],accel_mss,speed_ms,0,blend_radius_m)
    movel([0.654385, -1.416828, -2.550839, -0.744722, 1.570796, 2.225181],accel_mss,speed_ms,0,blend_radius_m)
    movel([0.655645, -1.417690, -2.550186, -0.744513, 1.570796, 2.226441],accel_mss,speed_ms,0,blend_radius_m)
    movel([0.656685, -1.418543, -2.549538, -0.744308, 1.570796, 2.227481],accel_mss,speed_ms,0,blend_radius_m)
    movel([0.655905, -1.418044, -2.549917, -0.744428, 1.570796, 2.226701],accel_mss,speed_ms,0,blend_radius_m)
    movel([0.654985, -1.417739, -2.550148, -0.744502, 1.570796, 2.225782],accel_mss,speed_ms,0,blend_radius_m)
    movel([0.653930, -1.417662, -2.550207, -0.744520, 1.570796, 2.224726],accel_mss,speed_ms,0,blend_radius_m)
    movel([0.652738, -1.417850, -2.550064, -0.744475, 1.570796, 2.223534],accel_mss,speed_ms,0,blend_radius_m)
    movel([0.651666, -1.418237, -2.549770, -0.744382, 1.570796, 2.222463],accel_mss,speed_ms,0,blend_radius_m)
    movel([0.650613, -1.418779, -2.549358, -0.744251, 1.570796, 2.221410],accel_mss,speed_ms,0,blend_radius_m)
    movel([0.649643, -1.419392, -2.548892, -0.744105, 1.570796, 2.220440],accel_mss,speed_ms,0,blend_radius_m)
    movel([0.648729, -1.420086, -2.548363, -0.743939, 1.570796, 2.219525],accel_mss,speed_ms,0,blend_radius_m)
    movel([0.647076, -1.421670, -2.547154, -0.743565, 1.570796, 2.217872],accel_mss,speed_ms,0,blend_radius_m)
    movel([0.645680, -1.423421, -2.545813, -0.743155, 1.570796, 2.216476],accel_mss,speed_ms,0,blend_radius_m)
    movel([0.644476, -1.425396, -2.544295, -0.742698, 1.570796, 2.215272],accel_mss,speed_ms,0,blend_radius_m)
    speed_ms = 0.005
    movel([0.644476, -1.416915, -2.540500, -0.754974, 1.570796, 2.215272],accel_mss,speed_ms,0,blend_radius_m)
    speed_ms = 0.040
    movel([0.649184, -1.413818, -2.542847, -0.755724, 1.570796, 2.219981],accel_mss,speed_ms,0,blend_radius_m)
    speed_ms = 0.005
    movel([0.649184, -1.422322, -2.546655, -0.743412, 1.570796, 2.219981],accel_mss,speed_ms,0,blend_radius_m)
    speed_ms = 0.025
    movel([0.648903, -1.422543, -2.546486, -0.743360, 1.570796, 2.219700],accel_mss,speed_ms,0,blend_radius_m)
    movel([0.648598, -1.422527, -2.546498, -0.743364, 1.570796, 2.219395],accel_mss,speed_ms,0,blend_radius_m)
    movel([0.648528, -1.422285, -2.546684, -0.743420, 1.570796, 2.219324],accel_mss,speed_ms,0,blend_radius_m)
    movel([0.648665, -1.421972, -2.546923, -0.743494, 1.570796, 2.219461],accel_mss,speed_ms,0,blend_radius_m)
    movel([0.649263, -1.421482, -2.547298, -0.743609, 1.570796, 2.220060],accel_mss,speed_ms,0,blend_radius_m)
    movel([0.649575, -1.421351, -2.547398, -0.743640, 1.570796, 2.220372],accel_mss,speed_ms,0,blend_radius_m)
    movel([0.649805, -1.421455, -2.547318, -0.743615, 1.570796, 2.220601],accel_mss,speed_ms,0,blend_radius_m)
    movel([0.649814, -1.421733, -2.547106, -0.743550, 1.570796, 2.220610],accel_mss,speed_ms,0,blend_radius_m)
    movel([0.649380, -1.422307, -2.546666, -0.743415, 1.570796, 2.220177],accel_mss,speed_ms,0,blend_radius_m)
    speed_ms = 0.005
    movel([0.649380, -1.413803, -2.542859, -0.755727, 1.570796, 2.220177],accel_mss,speed_ms,0,blend_radius_m)
    speed_ms = 0.040
    movel([0.644877, -1.421865, -2.536719, -0.753805, 1.570796, 2.215673],accel_mss,speed_ms,0,blend_radius_m)
    speed_ms = 0.005
    movel([0.644877, -1.430308, -2.540493, -0.741588, 1.570796, 2.215673],accel_mss,speed_ms,0,blend_radius_m)
    speed_ms = 0.025
    movel([0.646228, -1.429676, -2.540984, -0.741729, 1.570796, 2.217025],accel_mss,speed_ms,0,blend_radius_m)
    movel([0.647479, -1.428899, -2.541587, -0.741903, 1.570796, 2.218275],accel_mss,speed_ms,0,blend_radius_m)
    movel([0.649990, -1.427329, -2.542803, -0.742257, 1.570796, 2.220786],accel_mss,speed_ms,0,blend_radius_m)
    movel([0.651879, -1.426482, -2.543457, -0.742450, 1.570796, 2.222676],accel_mss,speed_ms,0,blend_radius_m)
    movel([0.657788, -1.424441, -2.545030, -0.742919, 1.570796, 2.228584],accel_mss,speed_ms,0,blend_radius_m)
    movel([0.658989, -1.423871, -2.545467, -0.743050, 1.570796, 2.229786],accel_mss,speed_ms,0,blend_radius_m)
    movel([0.659479, -1.423475, -2.545772, -0.743143, 1.570796, 2.230276],accel_mss,speed_ms,0,blend_radius_m)
    movel([0.659777, -1.422996, -2.546139, -0.743254, 1.570796, 2.230574],accel_mss,speed_ms,0,blend_radius_m)
    movel([0.659769, -1.422425, -2.546576, -0.743387, 1.570796, 2.230566],accel_mss,speed_ms,0,blend_radius_m)
    movel([0.659492, -1.421965, -2.546929, -0.743495, 1.570796, 2.230288],accel_mss,speed_ms,0,blend_radius_m)
    movel([0.658947, -1.421394, -2.547365, -0.743630, 1.570796, 2.229744],accel_mss,speed_ms,0,blend_radius_m)
    movel([0.658295, -1.421032, -2.547641, -0.743715, 1.570796, 2.229091],accel_mss,speed_ms,0,blend_radius_m)
    movel([0.657480, -1.420873, -2.547763, -0.743753, 1.570796, 2.228276],accel_mss,speed_ms,0,blend_radius_m)
    movel([0.656449, -1.420910, -2.547735, -0.743744, 1.570796, 2.227245],accel_mss,speed_ms,0,blend_radius_m)
    movel([0.655264, -1.421153, -2.547549, -0.743687, 1.570796, 2.226060],accel_mss,speed_ms,0,blend_radius_m)
    movel([0.654014, -1.421592, -2.547214, -0.743583, 1.570796, 2.224810],accel_mss,speed_ms,0,blend_radius_m)
    movel([0.652729, -1.422184, -2.546761, -0.743444, 1.570796, 2.223525],accel_mss,speed_ms,0,blend_radius_m)
    movel([0.651431, -1.422893, -2.546218, -0.743278, 1.570796, 2.222227],accel_mss,speed_ms,0,blend_radius_m)
    movel([0.648915, -1.424490, -2.544992, -0.742907, 1.570796, 2.219711],accel_mss,speed_ms,0,blend_radius_m)
    movel([0.646678, -1.426064, -2.543780, -0.742545, 1.570796, 2.217474],accel_mss,speed_ms,0,blend_radius_m)
    movel([0.642614, -1.429086, -2.541442, -0.741861, 1.570796, 2.213410],accel_mss,speed_ms,0,blend_radius_m)
    movel([0.641217, -1.430012, -2.540723, -0.741654, 1.570796, 2.212013],accel_mss,speed_ms,0,blend_radius_m)
    movel([0.639755, -1.430829, -2.540087, -0.741473, 1.570796, 2.210551],accel_mss,speed_ms,0,blend_radius_m)
    movel([0.638252, -1.431473, -2.539586, -0.741330, 1.570796, 2.209049],accel_mss,speed_ms,0,blend_radius_m)
    movel([0.636769, -1.431875, -2.539272, -0.741242, 1.570796, 2.207566],accel_mss,speed_ms,0,blend_radius_m)
    movel([0.635365, -1.431969, -2.539199, -0.741221, 1.570796, 2.206162],accel_mss,speed_ms,0,blend_radius_m)
    movel([0.636219, -1.432324, -2.538922, -0.741143, 1.570796, 2.207016],accel_mss,speed_ms,0,blend_radius_m)
    movel([0.637153, -1.432573, -2.538727, -0.741089, 1.570796, 2.207950],accel_mss,speed_ms,0,blend_radius_m)
    movel([0.638159, -1.432712, -2.538619, -0.741058, 1.570796, 2.208955],accel_mss,speed_ms,0,blend_radius_m)
    movel([0.639218, -1.432740, -2.538596, -0.741052, 1.570796, 2.210014],accel_mss,speed_ms,0,blend_radius_m)
    movel([0.638520, -1.433919, -2.537675, -0.740796, 1.570796, 2.209316],accel_mss,speed_ms,0,blend_radius_m)
    movel([0.637653, -1.435054, -2.536785, -0.740551, 1.570796, 2.208449],accel_mss,speed_ms,0,blend_radius_m)
    movel([0.636642, -1.436119, -2.535948, -0.740322, 1.570796, 2.207438],accel_mss,speed_ms,0,blend_radius_m)
    movel([0.635508, -1.437089, -2.535184, -0.740116, 1.570796, 2.206304],accel_mss,speed_ms,0,blend_radius_m)
    movel([0.637021, -1.436449, -2.535688, -0.740252, 1.570796, 2.207818],accel_mss,speed_ms,0,blend_radius_m)
    movel([0.638475, -1.435651, -2.536316, -0.740422, 1.570796, 2.209271],accel_mss,speed_ms,0,blend_radius_m)
    movel([0.639868, -1.434716, -2.537050, -0.740623, 1.570796, 2.210664],accel_mss,speed_ms,0,blend_radius_m)
    movel([0.641204, -1.433667, -2.537872, -0.740850, 1.570796, 2.212000],accel_mss,speed_ms,0,blend_radius_m)
    movel([0.640775, -1.434467, -2.537245, -0.740677, 1.570796, 2.211571],accel_mss,speed_ms,0,blend_radius_m)
    movel([0.640145, -1.435303, -2.536589, -0.740497, 1.570796, 2.210942],accel_mss,speed_ms,0,blend_radius_m)
    movel([0.636793, -1.438812, -2.533824, -0.739753, 1.570796, 2.207590],accel_mss,speed_ms,0,blend_radius_m)
    movel([0.636040, -1.439697, -2.533123, -0.739568, 1.570796, 2.206837],accel_mss,speed_ms,0,blend_radius_m)
    movel([0.635442, -1.440567, -2.532434, -0.739388, 1.570796, 2.206238],accel_mss,speed_ms,0,blend_radius_m)
    movel([0.636724, -1.439441, -2.533327, -0.739622, 1.570796, 2.207520],accel_mss,speed_ms,0,blend_radius_m)
    movel([0.638005, -1.438470, -2.534094, -0.739825, 1.570796, 2.208801],accel_mss,speed_ms,0,blend_radius_m)
    movel([0.640578, -1.436842, -2.535379, -0.740168, 1.570796, 2.211374],accel_mss,speed_ms,0,blend_radius_m)
    movel([0.643201, -1.435348, -2.536554, -0.740487, 1.570796, 2.213998],accel_mss,speed_ms,0,blend_radius_m)
    movel([0.645926, -1.433653, -2.537883, -0.740853, 1.570796, 2.216722],accel_mss,speed_ms,0,blend_radius_m)
    movel([0.647510, -1.432448, -2.538825, -0.741116, 1.570796, 2.218306],accel_mss,speed_ms,0,blend_radius_m)
    movel([0.648453, -1.431852, -2.539290, -0.741247, 1.570796, 2.219250],accel_mss,speed_ms,0,blend_radius_m)
    movel([0.648851, -1.431691, -2.539416, -0.741282, 1.570796, 2.219647],accel_mss,speed_ms,0,blend_radius_m)
    movel([0.649160, -1.431671, -2.539432, -0.741287, 1.570796, 2.219957],accel_mss,speed_ms,0,blend_radius_m)
    movel([0.649355, -1.431804, -2.539328, -0.741258, 1.570796, 2.220151],accel_mss,speed_ms,0,blend_radius_m)
    movel([0.649443, -1.432056, -2.539131, -0.741202, 1.570796, 2.220239],accel_mss,speed_ms,0,blend_radius_m)
    movel([0.649367, -1.432776, -2.538568, -0.741044, 1.570796, 2.220164],accel_mss,speed_ms,0,blend_radius_m)
    movel([0.649054, -1.433558, -2.537957, -0.740874, 1.570796, 2.219850],accel_mss,speed_ms,0,blend_radius_m)
    movel([0.648620, -1.434127, -2.537512, -0.740751, 1.570796, 2.219417],accel_mss,speed_ms,0,blend_radius_m)
    movel([0.650492, -1.432463, -2.538813, -0.741113, 1.570796, 2.221288],accel_mss,speed_ms,0,blend_radius_m)
    movel([0.652210, -1.430675, -2.540207, -0.741507, 1.570796, 2.223006],accel_mss,speed_ms,0,blend_radius_m)
    movel([0.653753, -1.428790, -2.541671, -0.741927, 1.570796, 2.224549],accel_mss,speed_ms,0,blend_radius_m)
    movel([0.655098, -1.426832, -2.543187, -0.742370, 1.570796, 2.225894],accel_mss,speed_ms,0,blend_radius_m)
    speed_ms = 0.005
    movel([0.655098, -1.418363, -2.539398, -0.754628, 1.570796, 2.225894],accel_mss,speed_ms,0,blend_radius_m)
    speed_ms = 0.040
    movel([0.656273, -1.420049, -2.538111, -0.754229, 1.570796, 2.227069],accel_mss,speed_ms,0,blend_radius_m)
    speed_ms = 0.005
    movel([0.656273, -1.428505, -2.541892, -0.741991, 1.570796, 2.227069],accel_mss,speed_ms,0,blend_radius_m)
    speed_ms = 0.025
    movel([0.657037, -1.429367, -2.541224, -0.741798, 1.570796, 2.227833],accel_mss,speed_ms,0,blend_radius_m)
    movel([0.657209, -1.429905, -2.540806, -0.741678, 1.570796, 2.228005],accel_mss,speed_ms,0,blend_radius_m)
    movel([0.657126, -1.430531, -2.540319, -0.741539, 1.570796, 2.227923],accel_mss,speed_ms,0,blend_radius_m)
    movel([0.656831, -1.431094, -2.539881, -0.741414, 1.570796, 2.227628],accel_mss,speed_ms,0,blend_radius_m)
    movel([0.650125, -1.439891, -2.532970, -0.739528, 1.570796, 2.220921],accel_mss,speed_ms,0,blend_radius_m)
    movel([0.649615, -1.440501, -2.532486, -0.739402, 1.570796, 2.220412],accel_mss,speed_ms,0,blend_radius_m)
    movel([0.649027, -1.441062, -2.532041, -0.739286, 1.570796, 2.219823],accel_mss,speed_ms,0,blend_radius_m)
    movel([0.648392, -1.441459, -2.531726, -0.739204, 1.570796, 2.219189],accel_mss,speed_ms,0,blend_radius_m)
    movel([0.647752, -1.441583, -2.531627, -0.739179, 1.570796, 2.218548],accel_mss,speed_ms,0,blend_radius_m)
    movel([0.647286, -1.441405, -2.531769, -0.739215, 1.570796, 2.218082],accel_mss,speed_ms,0,blend_radius_m)
    movel([0.646586, -1.440749, -2.532289, -0.739350, 1.570796, 2.217382],accel_mss,speed_ms,0,blend_radius_m)
    movel([0.646108, -1.440597, -2.532410, -0.739382, 1.570796, 2.216904],accel_mss,speed_ms,0,blend_radius_m)
    movel([0.645368, -1.440782, -2.532264, -0.739344, 1.570796, 2.216164],accel_mss,speed_ms,0,blend_radius_m)
    movel([0.644608, -1.441155, -2.531967, -0.739267, 1.570796, 2.215405],accel_mss,speed_ms,0,blend_radius_m)
    movel([0.643699, -1.441518, -2.531678, -0.739192, 1.570796, 2.214496],accel_mss,speed_ms,0,blend_radius_m)
    movel([0.642798, -1.441723, -2.531515, -0.739150, 1.570796, 2.213595],accel_mss,speed_ms,0,blend_radius_m)
    movel([0.641935, -1.441776, -2.531473, -0.739139, 1.570796, 2.212731],accel_mss,speed_ms,0,blend_radius_m)
    movel([0.641134, -1.441682, -2.531548, -0.739159, 1.570796, 2.211931],accel_mss,speed_ms,0,blend_radius_m)
    movel([0.640423, -1.441448, -2.531735, -0.739207, 1.570796, 2.211219],accel_mss,speed_ms,0,blend_radius_m)
    movel([0.639832, -1.441078, -2.532029, -0.739283, 1.570796, 2.210629],accel_mss,speed_ms,0,blend_radius_m)
    movel([0.639385, -1.440582, -2.532422, -0.739385, 1.570796, 2.210182],accel_mss,speed_ms,0,blend_radius_m)
    movel([0.639114, -1.439959, -2.532916, -0.739514, 1.570796, 2.209910],accel_mss,speed_ms,0,blend_radius_m)
    speed_ms = 0.005
    movel([0.639114, -1.431591, -2.529183, -0.751615, 1.570796, 2.209910],accel_mss,speed_ms,0,blend_radius_m)
    speed_ms = 0.040
    movel([0.629566, -1.437668, -2.524402, -0.750318, 1.570796, 2.200362],accel_mss,speed_ms,0,blend_radius_m)
    speed_ms = 0.005
    movel([0.629566, -1.445989, -2.528110, -0.738290, 1.570796, 2.200362],accel_mss,speed_ms,0,blend_radius_m)
    speed_ms = 0.025
    movel([0.624482, -1.455129, -2.520718, -0.736542, 1.570796, 2.195278],accel_mss,speed_ms,0,blend_radius_m)
    movel([0.623759, -1.456220, -2.519827, -0.736342, 1.570796, 2.194556],accel_mss,speed_ms,0,blend_radius_m)
    movel([0.623285, -1.456679, -2.519452, -0.736258, 1.570796, 2.194081],accel_mss,speed_ms,0,blend_radius_m)
    movel([0.622719, -1.457000, -2.519189, -0.736200, 1.570796, 2.193515],accel_mss,speed_ms,0,blend_radius_m)
    movel([0.621425, -1.457352, -2.518901, -0.736136, 1.570796, 2.192221],accel_mss,speed_ms,0,blend_radius_m)
    movel([0.620864, -1.457799, -2.518534, -0.736056, 1.570796, 2.191661],accel_mss,speed_ms,0,blend_radius_m)
    movel([0.620463, -1.458373, -2.518064, -0.735953, 1.570796, 2.191259],accel_mss,speed_ms,0,blend_radius_m)
    movel([0.620070, -1.459371, -2.517243, -0.735774, 1.570796, 2.190867],accel_mss,speed_ms,0,blend_radius_m)
    movel([0.619927, -1.460382, -2.516412, -0.735596, 1.570796, 2.190723],accel_mss,speed_ms,0,blend_radius_m)
    movel([0.619862, -1.462310, -2.514820, -0.735259, 1.570796, 2.190659],accel_mss,speed_ms,0,blend_radius_m)
    movel([0.619585, -1.463630, -2.513727, -0.735032, 1.570796, 2.190381],accel_mss,speed_ms,0,blend_radius_m)
    movel([0.618938, -1.465519, -2.512159, -0.734712, 1.570796, 2.189734],accel_mss,speed_ms,0,blend_radius_m)
    movel([0.618503, -1.466353, -2.511464, -0.734572, 1.570796, 2.189299],accel_mss,speed_ms,0,blend_radius_m)
    movel([0.618001, -1.466949, -2.510967, -0.734473, 1.570796, 2.188798],accel_mss,speed_ms,0,blend_radius_m)
    movel([0.617730, -1.467114, -2.510829, -0.734446, 1.570796, 2.188526],accel_mss,speed_ms,0,blend_radius_m)
    movel([0.617446, -1.467173, -2.510780, -0.734436, 1.570796, 2.188242],accel_mss,speed_ms,0,blend_radius_m)
    movel([0.617150, -1.467109, -2.510834, -0.734446, 1.570796, 2.187946],accel_mss,speed_ms,0,blend_radius_m)
    movel([0.616845, -1.466904, -2.511005, -0.734480, 1.570796, 2.187641],accel_mss,speed_ms,0,blend_radius_m)
    movel([0.616369, -1.467578, -2.510442, -0.734369, 1.570796, 2.187165],accel_mss,speed_ms,0,blend_radius_m)
    movel([0.616008, -1.468390, -2.509763, -0.734236, 1.570796, 2.186804],accel_mss,speed_ms,0,blend_radius_m)
    movel([0.615555, -1.470239, -2.508214, -0.733936, 1.570796, 2.186351],accel_mss,speed_ms,0,blend_radius_m)
    movel([0.615357, -1.472073, -2.506672, -0.733644, 1.570796, 2.186154],accel_mss,speed_ms,0,blend_radius_m)
    movel([0.615291, -1.473520, -2.505452, -0.733417, 1.570796, 2.186088],accel_mss,speed_ms,0,blend_radius_m)
    movel([0.615441, -1.475063, -2.504147, -0.733179, 1.570796, 2.186237],accel_mss,speed_ms,0,blend_radius_m)
    movel([0.615759, -1.476614, -2.502832, -0.732943, 1.570796, 2.186556],accel_mss,speed_ms,0,blend_radius_m)
    movel([0.615875, -1.478202, -2.501481, -0.732706, 1.570796, 2.186672],accel_mss,speed_ms,0,blend_radius_m)
    movel([0.615743, -1.479016, -2.500787, -0.732586, 1.570796, 2.186540],accel_mss,speed_ms,0,blend_radius_m)
    movel([0.615421, -1.479850, -2.500076, -0.732464, 1.570796, 2.186217],accel_mss,speed_ms,0,blend_radius_m)
    movel([0.615143, -1.480267, -2.499719, -0.732403, 1.570796, 2.185940],accel_mss,speed_ms,0,blend_radius_m)
    movel([0.614767, -1.480641, -2.499399, -0.732349, 1.570796, 2.185563],accel_mss,speed_ms,0,blend_radius_m)
    movel([0.614354, -1.480878, -2.499196, -0.732315, 1.570796, 2.185150],accel_mss,speed_ms,0,blend_radius_m)
    movel([0.613964, -1.480890, -2.499186, -0.732313, 1.570796, 2.184760],accel_mss,speed_ms,0,blend_radius_m)
    movel([0.613760, -1.480715, -2.499336, -0.732338, 1.570796, 2.184557],accel_mss,speed_ms,0,blend_radius_m)
    movel([0.613656, -1.480463, -2.499551, -0.732375, 1.570796, 2.184453],accel_mss,speed_ms,0,blend_radius_m)
    movel([0.613063, -1.477851, -2.501780, -0.732758, 1.570796, 2.183860],accel_mss,speed_ms,0,blend_radius_m)
    movel([0.612918, -1.476478, -2.502947, -0.732964, 1.570796, 2.183714],accel_mss,speed_ms,0,blend_radius_m)
    movel([0.612878, -1.475065, -2.504146, -0.733178, 1.570796, 2.183674],accel_mss,speed_ms,0,blend_radius_m)
    movel([0.612419, -1.475366, -2.503891, -0.733132, 1.570796, 2.183216],accel_mss,speed_ms,0,blend_radius_m)
    movel([0.612028, -1.475740, -2.503573, -0.733075, 1.570796, 2.182824],accel_mss,speed_ms,0,blend_radius_m)
    movel([0.611430, -1.476666, -2.502787, -0.732935, 1.570796, 2.182227],accel_mss,speed_ms,0,blend_radius_m)
    movel([0.611042, -1.477762, -2.501856, -0.732771, 1.570796, 2.181838],accel_mss,speed_ms,0,blend_radius_m)
    movel([0.610826, -1.478948, -2.500845, -0.732596, 1.570796, 2.181622],accel_mss,speed_ms,0,blend_radius_m)
    movel([0.610731, -1.481288, -2.498845, -0.732256, 1.570796, 2.181528],accel_mss,speed_ms,0,blend_radius_m)
    movel([0.610820, -1.483067, -2.497319, -0.732003, 1.570796, 2.181616],accel_mss,speed_ms,0,blend_radius_m)
    movel([0.610778, -1.483746, -2.496735, -0.731908, 1.570796, 2.181574],accel_mss,speed_ms,0,blend_radius_m)
    movel([0.610645, -1.484082, -2.496446, -0.731861, 1.570796, 2.181441],accel_mss,speed_ms,0,blend_radius_m)
    movel([0.610384, -1.484388, -2.496182, -0.731819, 1.570796, 2.181181],accel_mss,speed_ms,0,blend_radius_m)
    movel([0.610011, -1.484627, -2.495976, -0.731786, 1.570796, 2.180807],accel_mss,speed_ms,0,blend_radius_m)
    movel([0.609698, -1.484694, -2.495918, -0.731777, 1.570796, 2.180495],accel_mss,speed_ms,0,blend_radius_m)
    movel([0.609210, -1.484500, -2.496086, -0.731803, 1.570796, 2.180006],accel_mss,speed_ms,0,blend_radius_m)
    movel([0.608588, -1.484138, -2.496398, -0.731854, 1.570796, 2.179384],accel_mss,speed_ms,0,blend_radius_m)
    movel([0.608354, -1.484199, -2.496345, -0.731845, 1.570796, 2.179151],accel_mss,speed_ms,0,blend_radius_m)
    movel([0.608059, -1.484440, -2.496137, -0.731812, 1.570796, 2.178855],accel_mss,speed_ms,0,blend_radius_m)
    movel([0.607831, -1.484776, -2.495847, -0.731765, 1.570796, 2.178627],accel_mss,speed_ms,0,blend_radius_m)
    movel([0.607540, -1.485617, -2.495122, -0.731650, 1.570796, 2.178336],accel_mss,speed_ms,0,blend_radius_m)
    movel([0.607317, -1.487165, -2.493784, -0.731441, 1.570796, 2.178114],accel_mss,speed_ms,0,blend_radius_m)
    movel([0.607067, -1.490393, -2.490980, -0.731016, 1.570796, 2.177864],accel_mss,speed_ms,0,blend_radius_m)
    movel([0.606894, -1.493587, -2.488190, -0.730612, 1.570796, 2.177690],accel_mss,speed_ms,0,blend_radius_m)
    movel([0.606763, -1.494250, -2.487609, -0.730530, 1.570796, 2.177559],accel_mss,speed_ms,0,blend_radius_m)
    movel([0.606487, -1.494923, -2.487018, -0.730448, 1.570796, 2.177283],accel_mss,speed_ms,0,blend_radius_m)
    movel([0.606041, -1.495494, -2.486517, -0.730379, 1.570796, 2.176838],accel_mss,speed_ms,0,blend_radius_m)
    movel([0.605751, -1.495705, -2.486331, -0.730353, 1.570796, 2.176547],accel_mss,speed_ms,0,blend_radius_m)
    movel([0.605086, -1.495899, -2.486161, -0.730330, 1.570796, 2.175882],accel_mss,speed_ms,0,blend_radius_m)
    movel([0.604813, -1.495863, -2.486192, -0.730334, 1.570796, 2.175609],accel_mss,speed_ms,0,blend_radius_m)
    movel([0.604396, -1.495580, -2.486441, -0.730368, 1.570796, 2.175192],accel_mss,speed_ms,0,blend_radius_m)
    movel([0.604131, -1.495116, -2.486849, -0.730424, 1.570796, 2.174927],accel_mss,speed_ms,0,blend_radius_m)
    movel([0.603992, -1.494579, -2.487320, -0.730490, 1.570796, 2.174788],accel_mss,speed_ms,0,blend_radius_m)
    movel([0.603563, -1.491248, -2.490235, -0.730906, 1.570796, 2.174360],accel_mss,speed_ms,0,blend_radius_m)
    movel([0.603337, -1.487825, -2.493211, -0.731352, 1.570796, 2.174133],accel_mss,speed_ms,0,blend_radius_m)
    movel([0.603320, -1.484316, -2.496244, -0.731829, 1.570796, 2.174117],accel_mss,speed_ms,0,blend_radius_m)
    movel([0.603515, -1.480728, -2.499325, -0.732336, 1.570796, 2.174312],accel_mss,speed_ms,0,blend_radius_m)
    movel([0.603673, -1.479373, -2.500483, -0.732533, 1.570796, 2.174470],accel_mss,speed_ms,0,blend_radius_m)
    movel([0.604054, -1.477986, -2.501666, -0.732738, 1.570796, 2.174850],accel_mss,speed_ms,0,blend_radius_m)
    movel([0.604445, -1.477158, -2.502370, -0.732861, 1.570796, 2.175241],accel_mss,speed_ms,0,blend_radius_m)
    movel([0.604935, -1.476340, -2.503064, -0.732984, 1.570796, 2.175732],accel_mss,speed_ms,0,blend_radius_m)
    movel([0.606078, -1.474727, -2.504431, -0.733230, 1.570796, 2.176875],accel_mss,speed_ms,0,blend_radius_m)
    movel([0.610693, -1.469097, -2.509172, -0.734120, 1.570796, 2.181490],accel_mss,speed_ms,0,blend_radius_m)
    movel([0.611871, -1.467453, -2.510546, -0.734389, 1.570796, 2.182668],accel_mss,speed_ms,0,blend_radius_m)
    movel([0.612764, -1.465916, -2.511828, -0.734645, 1.570796, 2.183560],accel_mss,speed_ms,0,blend_radius_m)
    movel([0.613060, -1.465219, -2.512408, -0.734762, 1.570796, 2.183856],accel_mss,speed_ms,0,blend_radius_m)
    movel([0.613226, -1.464587, -2.512933, -0.734869, 1.570796, 2.184023],accel_mss,speed_ms,0,blend_radius_m)
    movel([0.613249, -1.464033, -2.513393, -0.734963, 1.570796, 2.184045],accel_mss,speed_ms,0,blend_radius_m)
    movel([0.613109, -1.463570, -2.513777, -0.735042, 1.570796, 2.183906],accel_mss,speed_ms,0,blend_radius_m)
    movel([0.612615, -1.462930, -2.514307, -0.735152, 1.570796, 2.183411],accel_mss,speed_ms,0,blend_radius_m)
    movel([0.612428, -1.462587, -2.514591, -0.735211, 1.570796, 2.183224],accel_mss,speed_ms,0,blend_radius_m)
    movel([0.612411, -1.462174, -2.514932, -0.735283, 1.570796, 2.183207],accel_mss,speed_ms,0,blend_radius_m)
    movel([0.612772, -1.461510, -2.515481, -0.735398, 1.570796, 2.183569],accel_mss,speed_ms,0,blend_radius_m)
    movel([0.613381, -1.460896, -2.515988, -0.735505, 1.570796, 2.184177],accel_mss,speed_ms,0,blend_radius_m)
    movel([0.615399, -1.458974, -2.517570, -0.735845, 1.570796, 2.186195],accel_mss,speed_ms,0,blend_radius_m)
    movel([0.617306, -1.456995, -2.519193, -0.736201, 1.570796, 2.188103],accel_mss,speed_ms,0,blend_radius_m)
    movel([0.619122, -1.454960, -2.520856, -0.736573, 1.570796, 2.189918],accel_mss,speed_ms,0,blend_radius_m)
    movel([0.620860, -1.452875, -2.522553, -0.736961, 1.570796, 2.191657],accel_mss,speed_ms,0,blend_radius_m)
    movel([0.624183, -1.448586, -2.526023, -0.737780, 1.570796, 2.194980],accel_mss,speed_ms,0,blend_radius_m)
    movel([0.627417, -1.444166, -2.529568, -0.738654, 1.570796, 2.198213],accel_mss,speed_ms,0,blend_radius_m)
    speed_ms = 0.005
    movel([0.627417, -1.435831, -2.525853, -0.750704, 1.570796, 2.198213],accel_mss,speed_ms,0,blend_radius_m)
    speed_ms = 0.040
    movel([0.617703, -1.446063, -2.517707, -0.748620, 1.570796, 2.188499],accel_mss,speed_ms,0,blend_radius_m)
    speed_ms = 0.005
    movel([0.617703, -1.454317, -2.521380, -0.736692, 1.570796, 2.188499],accel_mss,speed_ms,0,blend_radius_m)
    speed_ms = 0.025
    movel([0.614220, -1.456040, -2.519974, -0.736375, 1.570796, 2.185017],accel_mss,speed_ms,0,blend_radius_m)
    movel([0.610716, -1.457622, -2.518679, -0.736087, 1.570796, 2.181513],accel_mss,speed_ms,0,blend_radius_m)
    movel([0.607196, -1.459065, -2.517495, -0.735829, 1.570796, 2.177992],accel_mss,speed_ms,0,blend_radius_m)
    movel([0.603671, -1.460362, -2.516428, -0.735599, 1.570796, 2.174468],accel_mss,speed_ms,0,blend_radius_m)
    movel([0.606791, -1.458463, -2.517990, -0.735936, 1.570796, 2.177587],accel_mss,speed_ms,0,blend_radius_m)
    movel([0.609822, -1.456386, -2.519691, -0.736312, 1.570796, 2.180619],accel_mss,speed_ms,0,blend_radius_m)
    movel([0.612746, -1.454144, -2.521521, -0.736724, 1.570796, 2.183542],accel_mss,speed_ms,0,blend_radius_m)
    movel([0.615543, -1.451749, -2.523466, -0.737173, 1.570796, 2.186340],accel_mss,speed_ms,0,blend_radius_m)
    movel([0.612639, -1.453118, -2.522356, -0.736916, 1.570796, 2.183435],accel_mss,speed_ms,0,blend_radius_m)
    movel([0.609722, -1.454378, -2.521330, -0.736681, 1.570796, 2.180518],accel_mss,speed_ms,0,blend_radius_m)
    movel([0.606793, -1.455529, -2.520391, -0.736468, 1.570796, 2.177589],accel_mss,speed_ms,0,blend_radius_m)
    movel([0.603861, -1.456566, -2.519544, -0.736279, 1.570796, 2.174657],accel_mss,speed_ms,0,blend_radius_m)
    movel([0.600601, -1.457644, -2.518662, -0.736084, 1.570796, 2.171397],accel_mss,speed_ms,0,blend_radius_m)
    movel([0.597364, -1.458897, -2.517633, -0.735859, 1.570796, 2.168160],accel_mss,speed_ms,0,blend_radius_m)
    movel([0.595768, -1.459689, -2.516982, -0.735718, 1.570796, 2.166565],accel_mss,speed_ms,0,blend_radius_m)
    movel([0.594229, -1.460623, -2.516212, -0.735553, 1.570796, 2.165025],accel_mss,speed_ms,0,blend_radius_m)
    movel([0.592805, -1.461704, -2.515321, -0.735364, 1.570796, 2.163602],accel_mss,speed_ms,0,blend_radius_m)
    movel([0.591552, -1.462929, -2.514307, -0.735152, 1.570796, 2.162348],accel_mss,speed_ms,0,blend_radius_m)
    movel([0.592804, -1.461262, -2.515686, -0.735441, 1.570796, 2.163600],accel_mss,speed_ms,0,blend_radius_m)
    movel([0.594211, -1.459598, -2.517057, -0.735734, 1.570796, 2.165007],accel_mss,speed_ms,0,blend_radius_m)
    movel([0.595752, -1.457957, -2.518405, -0.736027, 1.570796, 2.166548],accel_mss,speed_ms,0,blend_radius_m)
    movel([0.597405, -1.456357, -2.519715, -0.736317, 1.570796, 2.168201],accel_mss,speed_ms,0,blend_radius_m)
    movel([0.599146, -1.454818, -2.520971, -0.736599, 1.570796, 2.169942],accel_mss,speed_ms,0,blend_radius_m)
    movel([0.600954, -1.453361, -2.522158, -0.736870, 1.570796, 2.171750],accel_mss,speed_ms,0,blend_radius_m)
    movel([0.602805, -1.452004, -2.523260, -0.737125, 1.570796, 2.173601],accel_mss,speed_ms,0,blend_radius_m)
    movel([0.604675, -1.450769, -2.524260, -0.737360, 1.570796, 2.175471],accel_mss,speed_ms,0,blend_radius_m)
    movel([0.601533, -1.452451, -2.522897, -0.737041, 1.570796, 2.172329],accel_mss,speed_ms,0,blend_radius_m)
    movel([0.598460, -1.454267, -2.521421, -0.736701, 1.570796, 2.169257],accel_mss,speed_ms,0,blend_radius_m)
    movel([0.595458, -1.456198, -2.519845, -0.736346, 1.570796, 2.166254],accel_mss,speed_ms,0,blend_radius_m)
    movel([0.592526, -1.458228, -2.518182, -0.735978, 1.570796, 2.163322],accel_mss,speed_ms,0,blend_radius_m)
    movel([0.589668, -1.460337, -2.516448, -0.735603, 1.570796, 2.160464],accel_mss,speed_ms,0,blend_radius_m)
    movel([0.586882, -1.462508, -2.514656, -0.735225, 1.570796, 2.157678],accel_mss,speed_ms,0,blend_radius_m)
    movel([0.581527, -1.466961, -2.510957, -0.734471, 1.570796, 2.152324],accel_mss,speed_ms,0,blend_radius_m)
    movel([0.583200, -1.465285, -2.512353, -0.734751, 1.570796, 2.153996],accel_mss,speed_ms,0,blend_radius_m)
    movel([0.584790, -1.463356, -2.513954, -0.735079, 1.570796, 2.155586],accel_mss,speed_ms,0,blend_radius_m)
    movel([0.587772, -1.459527, -2.517115, -0.735747, 1.570796, 2.158569],accel_mss,speed_ms,0,blend_radius_m)
    movel([0.589223, -1.457899, -2.518453, -0.736038, 1.570796, 2.160019],accel_mss,speed_ms,0,blend_radius_m)
    movel([0.590627, -1.456498, -2.519600, -0.736291, 1.570796, 2.161423],accel_mss,speed_ms,0,blend_radius_m)
    movel([0.593740, -1.453771, -2.521825, -0.736794, 1.570796, 2.164536],accel_mss,speed_ms,0,blend_radius_m)
    movel([0.593201, -1.454066, -2.521585, -0.736739, 1.570796, 2.163998],accel_mss,speed_ms,0,blend_radius_m)
    movel([0.592392, -1.454326, -2.521373, -0.736690, 1.570796, 2.163188],accel_mss,speed_ms,0,blend_radius_m)
    movel([0.588113, -1.455156, -2.520696, -0.736537, 1.570796, 2.158910],accel_mss,speed_ms,0,blend_radius_m)
    movel([0.586531, -1.455538, -2.520385, -0.736467, 1.570796, 2.157327],accel_mss,speed_ms,0,blend_radius_m)
    movel([0.584569, -1.456412, -2.519671, -0.736307, 1.570796, 2.155365],accel_mss,speed_ms,0,blend_radius_m)
    movel([0.582619, -1.457507, -2.518774, -0.736108, 1.570796, 2.153415],accel_mss,speed_ms,0,blend_radius_m)
    movel([0.578875, -1.459968, -2.516752, -0.735669, 1.570796, 2.149671],accel_mss,speed_ms,0,blend_radius_m)
    movel([0.580598, -1.458430, -2.518017, -0.735942, 1.570796, 2.151394],accel_mss,speed_ms,0,blend_radius_m)
    movel([0.582217, -1.456797, -2.519355, -0.736237, 1.570796, 2.153013],accel_mss,speed_ms,0,blend_radius_m)
    movel([0.585431, -1.453485, -2.522057, -0.736847, 1.570796, 2.156227],accel_mss,speed_ms,0,blend_radius_m)
    movel([0.587232, -1.451864, -2.523373, -0.737152, 1.570796, 2.158029],accel_mss,speed_ms,0,blend_radius_m)
    movel([0.589151, -1.450323, -2.524621, -0.737445, 1.570796, 2.159948],accel_mss,speed_ms,0,blend_radius_m)
    movel([0.593248, -1.447424, -2.526958, -0.738007, 1.570796, 2.164045],accel_mss,speed_ms,0,blend_radius_m)
    movel([0.601686, -1.442016, -2.531283, -0.739090, 1.570796, 2.172482],accel_mss,speed_ms,0,blend_radius_m)
    movel([0.599268, -1.442212, -2.531127, -0.739050, 1.570796, 2.170065],accel_mss,speed_ms,0,blend_radius_m)
    movel([0.596800, -1.442588, -2.530827, -0.738974, 1.570796, 2.167597],accel_mss,speed_ms,0,blend_radius_m)
    movel([0.594296, -1.443134, -2.530392, -0.738863, 1.570796, 2.165092],accel_mss,speed_ms,0,blend_radius_m)
    movel([0.591774, -1.443847, -2.529824, -0.738719, 1.570796, 2.162570],accel_mss,speed_ms,0,blend_radius_m)
    movel([0.589252, -1.444721, -2.529125, -0.738543, 1.570796, 2.160048],accel_mss,speed_ms,0,blend_radius_m)
    movel([0.586742, -1.445753, -2.528299, -0.738337, 1.570796, 2.157539],accel_mss,speed_ms,0,blend_radius_m)
    movel([0.584263, -1.446932, -2.527353, -0.738104, 1.570796, 2.155060],accel_mss,speed_ms,0,blend_radius_m)
    movel([0.581830, -1.448255, -2.526289, -0.737845, 1.570796, 2.152627],accel_mss,speed_ms,0,blend_radius_m)
    movel([0.582525, -1.447792, -2.526662, -0.737935, 1.570796, 2.153321],accel_mss,speed_ms,0,blend_radius_m)
    movel([0.583240, -1.447212, -2.527128, -0.738049, 1.570796, 2.154036],accel_mss,speed_ms,0,blend_radius_m)
    movel([0.584694, -1.445834, -2.528234, -0.738321, 1.570796, 2.155491],accel_mss,speed_ms,0,blend_radius_m)
    movel([0.587424, -1.443136, -2.530391, -0.738862, 1.570796, 2.158220],accel_mss,speed_ms,0,blend_radius_m)
    movel([0.589964, -1.441002, -2.532089, -0.739298, 1.570796, 2.160760],accel_mss,speed_ms,0,blend_radius_m)
    movel([0.592572, -1.438953, -2.533713, -0.739724, 1.570796, 2.163369],accel_mss,speed_ms,0,blend_radius_m)
    movel([0.595245, -1.436986, -2.535265, -0.740138, 1.570796, 2.166041],accel_mss,speed_ms,0,blend_radius_m)
    movel([0.597975, -1.435098, -2.536750, -0.740541, 1.570796, 2.168772],accel_mss,speed_ms,0,blend_radius_m)
    movel([0.600763, -1.433280, -2.538175, -0.740934, 1.570796, 2.171559],accel_mss,speed_ms,0,blend_radius_m)
    movel([0.603602, -1.431531, -2.539540, -0.741318, 1.570796, 2.174399],accel_mss,speed_ms,0,blend_radius_m)
    movel([0.609428, -1.428210, -2.542121, -0.742058, 1.570796, 2.180224],accel_mss,speed_ms,0,blend_radius_m)
    movel([0.607327, -1.428865, -2.541613, -0.741911, 1.570796, 2.178123],accel_mss,speed_ms,0,blend_radius_m)
    movel([0.601055, -1.430361, -2.540452, -0.741577, 1.570796, 2.171851],accel_mss,speed_ms,0,blend_radius_m)
    movel([0.598948, -1.430939, -2.540001, -0.741448, 1.570796, 2.169745],accel_mss,speed_ms,0,blend_radius_m)
    movel([0.596838, -1.431670, -2.539432, -0.741287, 1.570796, 2.167634],accel_mss,speed_ms,0,blend_radius_m)
    movel([0.594769, -1.432599, -2.538707, -0.741083, 1.570796, 2.165565],accel_mss,speed_ms,0,blend_radius_m)
    movel([0.592779, -1.433776, -2.537787, -0.740827, 1.570796, 2.163576],accel_mss,speed_ms,0,blend_radius_m)
    movel([0.595779, -1.431504, -2.539561, -0.741324, 1.570796, 2.166575],accel_mss,speed_ms,0,blend_radius_m)
    movel([0.598829, -1.429078, -2.541448, -0.741863, 1.570796, 2.169625],accel_mss,speed_ms,0,blend_radius_m)
    movel([0.601939, -1.426743, -2.543256, -0.742390, 1.570796, 2.172735],accel_mss,speed_ms,0,blend_radius_m)
    movel([0.603516, -1.425689, -2.544069, -0.742631, 1.570796, 2.174312],accel_mss,speed_ms,0,blend_radius_m)
    movel([0.605110, -1.424755, -2.544788, -0.742846, 1.570796, 2.175906],accel_mss,speed_ms,0,blend_radius_m)
    movel([0.610674, -1.421976, -2.546920, -0.743493, 1.570796, 2.181470],accel_mss,speed_ms,0,blend_radius_m)
    movel([0.616281, -1.419292, -2.548968, -0.744129, 1.570796, 2.187077],accel_mss,speed_ms,0,blend_radius_m)
    movel([0.612807, -1.419908, -2.548499, -0.743982, 1.570796, 2.183604],accel_mss,speed_ms,0,blend_radius_m)
    movel([0.609513, -1.420785, -2.547830, -0.743774, 1.570796, 2.180309],accel_mss,speed_ms,0,blend_radius_m)
    movel([0.606185, -1.421997, -2.546904, -0.743488, 1.570796, 2.176982],accel_mss,speed_ms,0,blend_radius_m)
    movel([0.602617, -1.423612, -2.545666, -0.743111, 1.570796, 2.173414],accel_mss,speed_ms,0,blend_radius_m)
    movel([0.604426, -1.422617, -2.546429, -0.743343, 1.570796, 2.175222],accel_mss,speed_ms,0,blend_radius_m)
    movel([0.606160, -1.421478, -2.547301, -0.743610, 1.570796, 2.176957],accel_mss,speed_ms,0,blend_radius_m)
    movel([0.612874, -1.416370, -2.551186, -0.744833, 1.570796, 2.183671],accel_mss,speed_ms,0,blend_radius_m)
    movel([0.614624, -1.415179, -2.552086, -0.745124, 1.570796, 2.185420],accel_mss,speed_ms,0,blend_radius_m)
    movel([0.616455, -1.414116, -2.552888, -0.745386, 1.570796, 2.187252],accel_mss,speed_ms,0,blend_radius_m)
    movel([0.618929, -1.412961, -2.553757, -0.745671, 1.570796, 2.189725],accel_mss,speed_ms,0,blend_radius_m)
    movel([0.620899, -1.412360, -2.554208, -0.745821, 1.570796, 2.191696],accel_mss,speed_ms,0,blend_radius_m)
    movel([0.621394, -1.412105, -2.554399, -0.745885, 1.570796, 2.192190],accel_mss,speed_ms,0,blend_radius_m)
    movel([0.621694, -1.411717, -2.554690, -0.745981, 1.570796, 2.192491],accel_mss,speed_ms,0,blend_radius_m)
    movel([0.621604, -1.411410, -2.554921, -0.746058, 1.570796, 2.192400],accel_mss,speed_ms,0,blend_radius_m)
    movel([0.621218, -1.411175, -2.555097, -0.746117, 1.570796, 2.192015],accel_mss,speed_ms,0,blend_radius_m)
    movel([0.620633, -1.411008, -2.555222, -0.746159, 1.570796, 2.191429],accel_mss,speed_ms,0,blend_radius_m)
    movel([0.619253, -1.410833, -2.555353, -0.746203, 1.570796, 2.190050],accel_mss,speed_ms,0,blend_radius_m)
    movel([0.618236, -1.410821, -2.555361, -0.746206, 1.570796, 2.189032],accel_mss,speed_ms,0,blend_radius_m)
    movel([0.620369, -1.409639, -2.556245, -0.746505, 1.570796, 2.191165],accel_mss,speed_ms,0,blend_radius_m)
    movel([0.622664, -1.408686, -2.556956, -0.746747, 1.570796, 2.193460],accel_mss,speed_ms,0,blend_radius_m)
    movel([0.627198, -1.407232, -2.558038, -0.747119, 1.570796, 2.197994],accel_mss,speed_ms,0,blend_radius_m)
    speed_ms = 0.005
    movel([0.627198, -1.398614, -2.554165, -0.759610, 1.570796, 2.197994],accel_mss,speed_ms,0,blend_radius_m)
    speed_ms = 0.040
    movel([0.620757, -1.396853, -2.555454, -0.760082, 1.570796, 2.191554],accel_mss,speed_ms,0,blend_radius_m)
    speed_ms = 0.005
    movel([0.620757, -1.405485, -2.559334, -0.747570, 1.570796, 2.191554],accel_mss,speed_ms,0,blend_radius_m)
    speed_ms = 0.025
    movel([0.620686, -1.404286, -2.560221, -0.747882, 1.570796, 2.191483],accel_mss,speed_ms,0,blend_radius_m)
    movel([0.620351, -1.403242, -2.560991, -0.748156, 1.570796, 2.191147],accel_mss,speed_ms,0,blend_radius_m)
    movel([0.619786, -1.402345, -2.561651, -0.748392, 1.570796, 2.190582],accel_mss,speed_ms,0,blend_radius_m)
    movel([0.619029, -1.401586, -2.562210, -0.748593, 1.570796, 2.189825],accel_mss,speed_ms,0,blend_radius_m)
    movel([0.618111, -1.400959, -2.562670, -0.748760, 1.570796, 2.188907],accel_mss,speed_ms,0,blend_radius_m)
    movel([0.617070, -1.400457, -2.563038, -0.748894, 1.570796, 2.187866],accel_mss,speed_ms,0,blend_radius_m)
    movel([0.614756, -1.399786, -2.563530, -0.749073, 1.570796, 2.185552],accel_mss,speed_ms,0,blend_radius_m)
    speed_ms = 0.005
    movel([0.614756, -1.391112, -2.559625, -0.761652, 1.570796, 2.185552],accel_mss,speed_ms,0,blend_radius_m)
    speed_ms = 0.040
    movel([0.625725, -1.390491, -2.560073, -0.761825, 1.570796, 2.196521],accel_mss,speed_ms,0,blend_radius_m)
    speed_ms = 0.005
    movel([0.625725, -1.399170, -2.563981, -0.749239, 1.570796, 2.196521],accel_mss,speed_ms,0,blend_radius_m)
    speed_ms = 0.025
    movel([0.626265, -1.397103, -2.565489, -0.749798, 1.570796, 2.197062],accel_mss,speed_ms,0,blend_radius_m)
    movel([0.626659, -1.395120, -2.566930, -0.750340, 1.570796, 2.197455],accel_mss,speed_ms,0,blend_radius_m)
    movel([0.626847, -1.393251, -2.568282, -0.750856, 1.570796, 2.197643],accel_mss,speed_ms,0,blend_radius_m)
    movel([0.626773, -1.391522, -2.569529, -0.751338, 1.570796, 2.197569],accel_mss,speed_ms,0,blend_radius_m)
    movel([0.626372, -1.389972, -2.570643, -0.751774, 1.570796, 2.197168],accel_mss,speed_ms,0,blend_radius_m)
    movel([0.625594, -1.388623, -2.571610, -0.752156, 1.570796, 2.196390],accel_mss,speed_ms,0,blend_radius_m)
    movel([0.624373, -1.387515, -2.572402, -0.752472, 1.570796, 2.195169],accel_mss,speed_ms,0,blend_radius_m)
    movel([0.623579, -1.387059, -2.572728, -0.752602, 1.570796, 2.194376],accel_mss,speed_ms,0,blend_radius_m)
    movel([0.622653, -1.386675, -2.573001, -0.752712, 1.570796, 2.193449],accel_mss,speed_ms,0,blend_radius_m)
    speed_ms = 0.005
    movel([0.622653, -1.377905, -2.569039, -0.765445, 1.570796, 2.193449],accel_mss,speed_ms,0,blend_radius_m)
    speed_ms = 0.040
    movel([0.631539, -1.377852, -2.569076, -0.765461, 1.570796, 2.202335],accel_mss,speed_ms,0,blend_radius_m)
    speed_ms = 0.005
    movel([0.631539, -1.386623, -2.573039, -0.752727, 1.570796, 2.202335],accel_mss,speed_ms,0,blend_radius_m)
    speed_ms = 0.025
    movel([0.633312, -1.382368, -2.576058, -0.753963, 1.570796, 2.204109],accel_mss,speed_ms,0,blend_radius_m)
    movel([0.633980, -1.380300, -2.577517, -0.754573, 1.570796, 2.204776],accel_mss,speed_ms,0,blend_radius_m)
    movel([0.634421, -1.378299, -2.578922, -0.755169, 1.570796, 2.205218],accel_mss,speed_ms,0,blend_radius_m)
    movel([0.634579, -1.376391, -2.580255, -0.755742, 1.570796, 2.205375],accel_mss,speed_ms,0,blend_radius_m)
    movel([0.634391, -1.374604, -2.581500, -0.756284, 1.570796, 2.205187],accel_mss,speed_ms,0,blend_radius_m)
    movel([0.633797, -1.372957, -2.582644, -0.756788, 1.570796, 2.204594],accel_mss,speed_ms,0,blend_radius_m)
    movel([0.632737, -1.371480, -2.583666, -0.757243, 1.570796, 2.203533],accel_mss,speed_ms,0,blend_radius_m)
    speed_ms = 0.005
    movel([0.632737, -1.362601, -2.579637, -0.770152, 1.570796, 2.203533],accel_mss,speed_ms,0,blend_radius_m)
    speed_ms = 0.040
    movel([0.638756, -1.366287, -2.577114, -0.768988, 1.570796, 2.209552],accel_mss,speed_ms,0,blend_radius_m)
    speed_ms = 0.005
    movel([0.638756, -1.375140, -2.581128, -0.756121, 1.570796, 2.209552],accel_mss,speed_ms,0,blend_radius_m)
    speed_ms = 0.025
    movel([0.640325, -1.372678, -2.582837, -0.756873, 1.570796, 2.211122],accel_mss,speed_ms,0,blend_radius_m)
    movel([0.641788, -1.370130, -2.584598, -0.757661, 1.570796, 2.212584],accel_mss,speed_ms,0,blend_radius_m)
    movel([0.643066, -1.367539, -2.586378, -0.758472, 1.570796, 2.213862],accel_mss,speed_ms,0,blend_radius_m)
    movel([0.644082, -1.364961, -2.588140, -0.759288, 1.570796, 2.214878],accel_mss,speed_ms,0,blend_radius_m)
    movel([0.644761, -1.362438, -2.589855, -0.760095, 1.570796, 2.215558],accel_mss,speed_ms,0,blend_radius_m)
    movel([0.644947, -1.361216, -2.590683, -0.760490, 1.570796, 2.215744],accel_mss,speed_ms,0,blend_radius_m)
    movel([0.644972, -1.358881, -2.592258, -0.761249, 1.570796, 2.215768],accel_mss,speed_ms,0,blend_radius_m)
    movel([0.644788, -1.357782, -2.592997, -0.761610, 1.570796, 2.215584],accel_mss,speed_ms,0,blend_radius_m)
    movel([0.644460, -1.356735, -2.593700, -0.761954, 1.570796, 2.215256],accel_mss,speed_ms,0,blend_radius_m)
    movel([0.643978, -1.355752, -2.594358, -0.762279, 1.570796, 2.214774],accel_mss,speed_ms,0,blend_radius_m)
    speed_ms = 0.005
    movel([0.643978, -1.346763, -2.590258, -0.775368, 1.570796, 2.214774],accel_mss,speed_ms,0,blend_radius_m)
    speed_ms = 0.040
    movel([0.650408, -1.350380, -2.587863, -0.774146, 1.570796, 2.221204],accel_mss,speed_ms,0,blend_radius_m)
    speed_ms = 0.005
    movel([0.650408, -1.359345, -2.591946, -0.761098, 1.570796, 2.221204],accel_mss,speed_ms,0,blend_radius_m)
    speed_ms = 0.025
    movel([0.652391, -1.356509, -2.593851, -0.762029, 1.570796, 2.223187],accel_mss,speed_ms,0,blend_radius_m)
    movel([0.654173, -1.353565, -2.595817, -0.763007, 1.570796, 2.224970],accel_mss,speed_ms,0,blend_radius_m)
    movel([0.655681, -1.350573, -2.597802, -0.764014, 1.570796, 2.226477],accel_mss,speed_ms,0,blend_radius_m)
    movel([0.656825, -1.347599, -2.599763, -0.765027, 1.570796, 2.227621],accel_mss,speed_ms,0,blend_radius_m)
    movel([0.657528, -1.344707, -2.601658, -0.766024, 1.570796, 2.228325],accel_mss,speed_ms,0,blend_radius_m)
    movel([0.657685, -1.343314, -2.602567, -0.766508, 1.570796, 2.228481],accel_mss,speed_ms,0,blend_radius_m)
    movel([0.657703, -1.341966, -2.603444, -0.766979, 1.570796, 2.228499],accel_mss,speed_ms,0,blend_radius_m)
    movel([0.657564, -1.340675, -2.604281, -0.767433, 1.570796, 2.228360],accel_mss,speed_ms,0,blend_radius_m)
    movel([0.657263, -1.339444, -2.605078, -0.767868, 1.570796, 2.228060],accel_mss,speed_ms,0,blend_radius_m)
    movel([0.656787, -1.338289, -2.605822, -0.768277, 1.570796, 2.227583],accel_mss,speed_ms,0,blend_radius_m)
    movel([0.656126, -1.337213, -2.606515, -0.768661, 1.570796, 2.226923],accel_mss,speed_ms,0,blend_radius_m)
    speed_ms = 0.005
    movel([0.656126, -1.328100, -2.602333, -0.781957, 1.570796, 2.226923],accel_mss,speed_ms,0,blend_radius_m)
    speed_ms = 0.040
    movel([0.621666, -1.319357, -2.607827, -0.785205, 1.570796, 2.192462],accel_mss,speed_ms,0,blend_radius_m)
    speed_ms = 0.005
    movel([0.621666, -1.328527, -2.612049, -0.771813, 1.570796, 2.192462],accel_mss,speed_ms,0,blend_radius_m)
    speed_ms = 0.025
    movel([0.622565, -1.330597, -2.610739, -0.771053, 1.570796, 2.193361],accel_mss,speed_ms,0,blend_radius_m)
    movel([0.623171, -1.332843, -2.609312, -0.770234, 1.570796, 2.193967],accel_mss,speed_ms,0,blend_radius_m)
    movel([0.623505, -1.335243, -2.607779, -0.769367, 1.570796, 2.194301],accel_mss,speed_ms,0,blend_radius_m)
    movel([0.623585, -1.337774, -2.606154, -0.768461, 1.570796, 2.194382],accel_mss,speed_ms,0,blend_radius_m)
    movel([0.623426, -1.340411, -2.604452, -0.767526, 1.570796, 2.194222],accel_mss,speed_ms,0,blend_radius_m)
    movel([0.623051, -1.343134, -2.602684, -0.766571, 1.570796, 2.193847],accel_mss,speed_ms,0,blend_radius_m)
    movel([0.622469, -1.345924, -2.600862, -0.765603, 1.570796, 2.193266],accel_mss,speed_ms,0,blend_radius_m)
    movel([0.621708, -1.348755, -2.599002, -0.764632, 1.570796, 2.192504],accel_mss,speed_ms,0,blend_radius_m)
    movel([0.620776, -1.351608, -2.597117, -0.763664, 1.570796, 2.191572],accel_mss,speed_ms,0,blend_radius_m)
    movel([0.619696, -1.354465, -2.595217, -0.762707, 1.570796, 2.190492],accel_mss,speed_ms,0,blend_radius_m)
    movel([0.618481, -1.357303, -2.593319, -0.761767, 1.570796, 2.189278],accel_mss,speed_ms,0,blend_radius_m)
    movel([0.617148, -1.360107, -2.591432, -0.760850, 1.570796, 2.187944],accel_mss,speed_ms,0,blend_radius_m)
    movel([0.615715, -1.362853, -2.589574, -0.759962, 1.570796, 2.186512],accel_mss,speed_ms,0,blend_radius_m)
    movel([0.614192, -1.365529, -2.587753, -0.759107, 1.570796, 2.184989],accel_mss,speed_ms,0,blend_radius_m)
    movel([0.612601, -1.368109, -2.585988, -0.758293, 1.570796, 2.183397],accel_mss,speed_ms,0,blend_radius_m)
    movel([0.610954, -1.370581, -2.584286, -0.757521, 1.570796, 2.181750],accel_mss,speed_ms,0,blend_radius_m)
    movel([0.608645, -1.373803, -2.582057, -0.756529, 1.570796, 2.179441],accel_mss,speed_ms,0,blend_radius_m)
    movel([0.605844, -1.377409, -2.579544, -0.755436, 1.570796, 2.176640],accel_mss,speed_ms,0,blend_radius_m)
    movel([0.602687, -1.381032, -2.577001, -0.754356, 1.570796, 2.173483],accel_mss,speed_ms,0,blend_radius_m)
